C09129=1128.647,-3.756,-49.814,179.578,6.251,149.256
C09130=1128.642,-3.507,-49.827,179.579,6.255,149.256
C09131=1128.636,-3.257,-49.840,179.579,6.260,149.257
C09132=1128.632,-3.007,-49.853,179.580,6.265,149.258
C09133=1128.627,-2.758,-49.866,179.581,6.269,149.259
C09134=1128.621,-2.508,-49.879,179.581,6.274,149.260
C09135=1128.616,-2.259,-49.891,179.582,6.278,149.260
C09136=1128.611,-2.009,-49.905,179.582,6.283,149.261
C09137=1128.605,-1.760,-49.918,179.583,6.287,149.262
C09138=1128.600,-1.510,-49.930,179.583,6.291,149.263
C09139=1128.595,-1.260,-49.944,179.584,6.296,149.264
C09140=1128.590,-1.011,-49.956,179.585,6.300,149.264
C09141=1128.585,-0.761,-49.969,179.585,6.305,149.265
C09142=1128.580,-0.511,-49.982,179.586,6.310,149.266
C09143=1128.575,-0.262,-49.996,179.586,6.314,149.267
C09144=1128.569,-0.012,-50.009,179.587,6.318,149.268
C09145=1128.564,0.237,-50.022,179.587,6.323,149.269
C09146=1128.559,0.487,-50.035,179.588,6.328,149.269
C09147=1128.554,0.737,-50.048,179.588,6.332,149.270
C09148=1128.549,0.986,-50.061,179.589,6.337,149.271
C09149=1128.543,1.235,-50.075,179.589,6.341,149.272
C09150=1128.539,1.485,-50.088,179.590,6.345,149.273
C09151=1128.534,1.735,-50.100,179.590,6.350,149.274
C09152=1128.528,1.985,-50.114,179.591,6.355,149.274
C09153=1128.523,2.234,-50.126,179.591,6.360,149.275
C09154=1128.518,2.483,-50.140,179.592,6.363,149.276
C09155=1128.513,2.733,-50.153,179.592,6.368,149.277
C09156=1128.507,2.983,-50.166,179.593,6.373,149.278
C09157=1128.503,3.233,-50.179,179.593,6.377,149.279
C09158=1128.497,3.482,-50.193,179.593,6.381,149.280
C09159=1128.492,3.731,-50.206,179.594,6.386,149.280
C09160=1128.487,3.982,-50.219,179.595,6.390,149.281
C09161=1128.482,4.230,-50.233,179.595,6.395,149.282
C09162=1128.477,4.481,-50.246,179.596,6.400,149.283
C09163=1128.472,4.730,-50.259,179.596,6.404,149.284
C09164=1128.466,4.980,-50.273,179.596,6.408,149.285
C09165=1128.462,5.229,-50.286,179.597,6.413,149.285
C09166=1128.456,5.479,-50.299,179.597,6.418,149.286
C09167=1128.452,5.728,-50.313,179.597,6.422,149.287
C09168=1128.446,5.978,-50.326,179.598,6.426,149.288
C09169=1128.441,6.228,-50.339,179.599,6.431,149.289
C09170=1128.436,6.477,-50.353,179.599,6.435,149.290
C09171=1128.431,6.693,-50.364,179.599,6.439,149.291
C09172=1128.427,6.908,-50.375,179.600,6.443,149.291
C09173=1128.423,7.123,-50.387,179.600,6.447,149.292
C09174=1128.418,7.339,-50.399,179.600,6.450,149.293
C09175=1128.413,7.555,-50.410,179.601,6.455,149.293
C09176=1128.409,7.770,-50.422,179.601,6.459,149.294
C09177=1128.405,7.985,-50.434,179.601,6.462,149.295
C09178=1128.401,8.200,-50.445,179.601,6.466,149.296
C09179=1128.395,8.450,-50.459,179.602,6.470,149.296
C09180=1128.390,8.700,-50.473,179.604,6.476,149.297
C09181=1128.385,8.949,-50.485,179.605,6.480,149.298
C09182=1128.380,9.199,-50.500,179.605,6.485,149.299
C09183=1128.375,9.448,-50.512,179.606,6.490,149.300
C09184=1128.370,9.698,-50.527,179.607,6.495,149.300
C09185=1128.364,9.947,-50.540,179.608,6.500,149.301
C09186=1128.360,10.197,-50.554,179.609,6.504,149.302
C09187=1128.354,10.447,-50.567,179.609,6.509,149.303
C09188=1128.349,10.696,-50.581,179.611,6.514,149.303
C09189=1128.344,10.946,-50.594,179.612,6.518,149.304
C09190=1128.339,11.195,-50.608,179.612,6.523,149.305
C09191=1128.334,11.446,-50.621,179.613,6.528,149.306
C09192=1128.328,11.695,-50.635,179.614,6.533,149.307
C09193=1128.324,11.944,-50.649,179.615,6.537,149.307
C09194=1128.318,12.194,-50.662,179.616,6.542,149.308
C09195=1128.313,12.443,-50.676,179.617,6.546,149.309
C09196=1128.308,12.693,-50.689,179.618,6.552,149.310
C09197=1128.303,12.942,-50.703,179.619,6.556,149.310
C09198=1128.298,13.192,-50.718,179.620,6.561,149.311
C09199=1128.292,13.442,-50.731,179.621,6.565,149.312
C09200=1128.288,13.691,-50.745,179.622,6.570,149.313
C09201=1128.283,13.941,-50.759,179.623,6.575,149.313
C09202=1128.277,14.190,-50.772,179.624,6.579,149.314
C09203=1128.272,14.440,-50.786,179.625,6.584,149.315
C09204=1128.267,14.689,-50.800,179.626,6.588,149.316
C09205=1128.262,14.939,-50.814,179.627,6.593,149.316
C09206=1128.257,15.189,-50.827,179.628,6.598,149.317
C09207=1128.252,15.438,-50.841,179.629,6.603,149.318
C09208=1128.247,15.688,-50.856,179.629,6.607,149.319
C09209=1128.242,15.937,-50.870,179.630,6.612,149.319
C09210=1128.236,16.187,-50.883,179.631,6.616,149.320
C09211=1128.232,16.436,-50.897,179.632,6.621,149.321
C09212=1128.227,16.686,-50.911,179.634,6.626,149.321
C09213=1128.221,16.935,-50.925,179.635,6.630,149.322
C09214=1128.216,17.185,-50.939,179.635,6.635,149.323
C09215=1128.211,17.435,-50.953,179.636,6.639,149.324
C09216=1128.205,17.684,-50.967,179.637,6.644,149.324
C09217=1128.200,17.934,-50.981,179.639,6.649,149.325
C09218=1128.195,18.184,-50.995,179.640,6.653,149.326
C09219=1128.191,18.432,-51.009,179.641,6.658,149.326
C09220=1128.186,18.682,-51.023,179.641,6.662,149.327
C09221=1128.181,18.932,-51.037,179.642,6.667,149.328
C09222=1128.176,19.181,-51.051,179.643,6.671,149.329
C09223=1128.170,19.431,-51.065,179.645,6.676,149.329
C09224=1128.165,19.681,-51.079,179.645,6.681,149.330
C09225=1128.160,19.930,-51.093,179.647,6.685,149.331
C09226=1128.155,20.180,-51.107,179.648,6.690,149.331
C09227=1128.151,20.395,-51.120,179.649,6.694,149.332
C09228=1128.146,20.610,-51.132,179.649,6.697,149.333
C09229=1128.142,20.826,-51.144,179.651,6.701,149.333
C09230=1128.137,21.041,-51.156,179.651,6.705,149.334
C09231=1128.133,21.256,-51.168,179.652,6.709,149.335
C09232=1128.128,21.471,-51.181,179.652,6.713,149.335
C09233=1128.124,21.687,-51.192,179.654,6.717,149.336
C09234=1128.120,21.902,-51.205,179.655,6.721,149.336
C09235=1128.115,22.151,-51.220,179.656,6.725,149.337
C09236=1128.110,22.401,-51.234,179.657,6.730,149.338
C09237=1128.105,22.651,-51.248,179.658,6.734,149.338
C09238=1128.099,22.900,-51.262,179.659,6.739,149.339
C09239=1128.094,23.149,-51.276,179.660,6.743,149.340
C09240=1128.089,23.399,-51.291,179.661,6.747,149.340
C09241=1128.084,23.649,-51.305,179.662,6.752,149.341
C09242=1128.079,23.899,-51.319,179.664,6.757,149.342
C09243=1128.074,24.148,-51.334,179.664,6.761,149.343
C09244=1128.069,24.397,-51.348,179.665,6.766,149.343
C09245=1128.063,24.647,-51.363,179.666,6.770,149.344
C09246=1128.058,24.896,-51.377,179.667,6.774,149.344
C09247=1128.054,25.146,-51.392,179.668,6.779,149.345
C09248=1128.049,25.396,-51.406,179.669,6.783,149.346
C09249=1128.044,25.646,-51.420,179.670,6.787,149.346
C09250=1128.038,25.894,-51.435,179.672,6.792,149.347
C09251=1128.033,26.144,-51.449,179.673,6.797,149.348
C09252=1128.028,26.393,-51.463,179.674,6.801,149.348
C09253=1128.023,26.643,-51.478,179.675,6.805,149.349
C09254=1128.018,26.893,-51.492,179.676,6.810,149.350
C09255=1128.013,27.142,-51.507,179.677,6.814,149.351
C09256=1128.008,27.392,-51.522,179.678,6.819,149.351
C09257=1128.003,27.642,-51.536,179.679,6.823,149.352
C09258=1127.998,27.890,-51.551,179.680,6.827,149.352
C09259=1127.992,28.140,-51.566,179.681,6.832,149.353
C09260=1127.987,28.390,-51.580,179.682,6.836,149.354
C09261=1127.982,28.639,-51.594,179.684,6.841,149.354
C09262=1127.978,28.889,-51.609,179.685,6.845,149.355
C09263=1127.972,29.139,-51.624,179.686,6.850,149.356
C09264=1127.967,29.388,-51.638,179.687,6.854,149.356
C09265=1127.962,29.637,-51.653,179.688,6.858,149.357
C09266=1127.958,29.887,-51.668,179.690,6.862,149.357
C09267=1127.953,30.136,-51.683,179.691,6.867,149.358
C09268=1127.947,30.386,-51.697,179.692,6.871,149.359
C09269=1127.942,30.636,-51.712,179.693,6.875,149.359
C09270=1127.938,30.885,-51.727,179.694,6.880,149.360
C09271=1127.932,31.135,-51.742,179.695,6.884,149.361
C09272=1127.927,31.384,-51.757,179.696,6.888,149.361
C09273=1127.922,31.634,-51.771,179.698,6.893,149.362
C09274=1127.917,31.884,-51.785,179.699,6.898,149.363
C09275=1127.912,32.133,-51.801,179.700,6.902,149.363
C09276=1127.907,32.383,-51.815,179.701,6.906,149.364
C09277=1127.902,32.632,-51.830,179.702,6.910,149.365
C09278=1127.897,32.882,-51.845,179.703,6.915,149.365
C09279=1127.892,33.131,-51.860,179.704,6.919,149.366
C09280=1127.887,33.381,-51.874,179.705,6.923,149.366
C09281=1127.882,33.630,-51.890,179.707,6.927,149.367
C09282=1127.877,33.880,-51.904,179.708,6.932,149.368
C09283=1127.872,34.095,-51.917,179.709,6.936,149.368
C09284=1127.867,34.310,-51.930,179.710,6.939,149.369
C09285=1127.863,34.525,-51.943,179.711,6.943,149.369
C09286=1127.860,34.740,-51.956,179.712,6.947,149.370
C09287=1127.855,34.955,-51.969,179.713,6.950,149.370
C09288=1127.850,35.170,-51.982,179.714,6.954,149.371
C09289=1127.846,35.386,-51.994,179.715,6.958,149.371
C09290=1127.841,35.601,-52.007,179.716,6.961,149.372
C09291=1127.837,35.850,-52.022,179.717,6.965,149.372
C09292=1127.831,36.100,-52.037,179.718,6.970,149.373
C09293=1127.827,36.349,-52.052,179.719,6.974,149.374
C09294=1127.821,36.599,-52.068,179.720,6.978,149.374
C09295=1127.816,36.848,-52.082,179.721,6.983,149.375
C09296=1127.811,37.098,-52.098,179.723,6.987,149.375
C09297=1127.806,37.347,-52.113,179.724,6.991,149.376
C09298=1127.801,37.596,-52.128,179.725,6.995,149.377
C09299=1127.796,37.846,-52.142,179.726,6.999,149.377
C09300=1127.791,38.096,-52.158,179.727,7.004,149.378
C09301=1127.786,38.345,-52.173,179.729,7.008,149.378
C09302=1127.781,38.595,-52.188,179.730,7.013,149.379
C09303=1127.776,38.844,-52.203,179.731,7.017,149.380
C09304=1127.771,39.094,-52.219,179.733,7.021,149.380
C09305=1127.766,39.343,-52.234,179.734,7.025,149.381
C09306=1127.760,39.593,-52.249,179.735,7.030,149.381
C09307=1127.756,39.842,-52.264,179.736,7.034,149.382
C09308=1127.751,40.092,-52.280,179.738,7.038,149.382
C09309=1127.746,40.341,-52.295,179.739,7.042,149.383
C09310=1127.741,40.590,-52.310,179.740,7.047,149.384
C09311=1127.735,40.840,-52.326,179.741,7.051,149.384
C09312=1127.730,41.090,-52.340,179.743,7.055,149.385
C09313=1127.725,41.339,-52.356,179.744,7.059,149.385
C09314=1127.720,41.588,-52.371,179.745,7.063,149.386
C09315=1127.716,41.838,-52.387,179.746,7.067,149.386
C09316=1127.710,42.088,-52.402,179.747,7.072,149.387
C09317=1127.706,42.337,-52.417,179.748,7.076,149.388
C09318=1127.700,42.586,-52.433,179.750,7.080,149.388
C09319=1127.696,42.835,-52.448,179.751,7.084,149.389
C09320=1127.691,43.085,-52.464,179.752,7.088,149.389
C09321=1127.685,43.335,-52.479,179.754,7.092,149.390
C09322=1127.680,43.584,-52.494,179.755,7.097,149.391
C09323=1127.675,43.834,-52.509,179.756,7.101,149.391
C09324=1127.670,44.083,-52.525,179.757,7.105,149.392
C09325=1127.666,44.333,-52.540,179.758,7.109,149.392
C09326=1127.660,44.582,-52.556,179.759,7.113,149.393
C09327=1127.655,44.832,-52.571,179.761,7.117,149.393
C09328=1127.650,45.081,-52.586,179.762,7.122,149.394
C09329=1127.645,45.331,-52.602,179.764,7.126,149.394
C09330=1127.640,45.580,-52.618,179.765,7.130,149.395
C09331=1127.635,45.829,-52.634,179.766,7.134,149.396
C09332=1127.630,46.078,-52.649,179.767,7.138,149.396
C09333=1127.626,46.328,-52.665,179.768,7.142,149.397
C09334=1127.620,46.578,-52.681,179.770,7.146,149.397
C09335=1127.615,46.827,-52.696,179.771,7.151,149.398
C09336=1127.611,47.077,-52.712,179.772,7.155,149.398
C09337=1127.605,47.326,-52.727,179.774,7.159,149.399
C09338=1127.600,47.576,-52.743,179.775,7.163,149.400
C09339=1127.596,47.791,-52.757,179.776,7.166,149.400
C09340=1127.592,48.006,-52.770,179.777,7.170,149.400
C09341=1127.588,48.221,-52.783,179.778,7.173,149.401
C09342=1127.583,48.436,-52.797,179.779,7.178,149.401
C09343=1127.579,48.652,-52.811,179.780,7.181,149.402
C09344=1127.574,48.866,-52.825,179.782,7.185,149.402
C09345=1127.570,49.082,-52.838,179.783,7.188,149.403
C09346=1127.566,49.297,-52.851,179.784,7.191,149.403
C09347=1127.561,49.545,-52.867,179.785,7.195,149.404
C09348=1127.556,49.796,-52.883,179.786,7.199,149.404
C09349=1127.550,50.045,-52.899,179.787,7.204,149.405
C09350=1127.546,50.294,-52.914,179.789,7.207,149.405
C09351=1127.541,50.544,-52.930,179.790,7.212,149.406
C09352=1127.536,50.793,-52.946,179.792,7.216,149.406
C09353=1127.531,51.043,-52.962,179.793,7.220,149.407
C09354=1127.526,51.292,-52.978,179.794,7.224,149.407
C09355=1127.521,51.541,-52.994,179.795,7.228,149.408
C09356=1127.516,51.791,-53.010,179.797,7.232,149.409
C09357=1127.510,52.041,-53.025,179.798,7.236,149.409
C09358=1127.505,52.290,-53.042,179.799,7.240,149.410
C09359=1127.501,52.539,-53.057,179.801,7.245,149.410
C09360=1127.496,52.789,-53.073,179.802,7.249,149.411
C09361=1127.491,53.038,-53.089,179.803,7.253,149.411
C09362=1127.486,53.288,-53.105,179.805,7.257,149.412
C09363=1127.481,53.537,-53.121,179.806,7.261,149.412
C09364=1127.476,53.787,-53.137,179.807,7.265,149.413
C09365=1127.471,54.036,-53.153,179.809,7.269,149.413
C09366=1127.466,54.285,-53.169,179.810,7.273,149.414
C09367=1127.461,54.535,-53.185,179.811,7.277,149.415
C09368=1127.456,54.784,-53.202,179.813,7.281,149.415
C09369=1127.451,55.034,-53.217,179.814,7.286,149.416
C09370=1127.446,55.283,-53.233,179.815,7.290,149.416
C09371=1127.441,55.533,-53.250,179.817,7.293,149.416
C09372=1127.436,55.782,-53.265,179.818,7.298,149.417
C09373=1127.431,56.031,-53.282,179.820,7.302,149.418
C09374=1127.426,56.281,-53.297,179.821,7.306,149.418
C09375=1127.422,56.530,-53.314,179.822,7.310,149.419
C09376=1127.416,56.780,-53.330,179.823,7.314,149.419
C09377=1127.411,57.030,-53.347,179.825,7.318,149.420
C09378=1127.406,57.278,-53.363,179.826,7.322,149.420
C09379=1127.401,57.528,-53.379,179.828,7.326,149.421
C09380=1127.396,57.777,-53.396,179.829,7.330,149.421
C09381=1127.391,58.027,-53.411,179.830,7.335,149.422
C09382=1127.386,58.276,-53.428,179.832,7.338,149.422
C09383=1127.381,58.526,-53.444,179.833,7.342,149.423
C09384=1127.376,58.775,-53.460,179.834,7.347,149.423
C09385=1127.372,59.024,-53.477,179.836,7.351,149.424
C09386=1127.366,59.274,-53.492,179.837,7.355,149.424
C09387=1127.361,59.524,-53.510,179.839,7.359,149.425
C09388=1127.356,59.772,-53.526,179.840,7.363,149.425
C09389=1127.351,60.023,-53.542,179.841,7.367,149.426
C09390=1127.346,60.271,-53.558,179.843,7.371,149.426
C09391=1127.342,60.521,-53.575,179.844,7.374,149.427
C09392=1127.336,60.770,-53.590,179.845,7.378,149.427
C09393=1127.331,61.020,-53.608,179.847,7.382,149.428
C09394=1127.327,61.269,-53.624,179.848,7.386,149.428
C09395=1127.322,61.484,-53.638,179.849,7.390,149.429
C09396=1127.318,61.699,-53.653,179.850,7.394,149.429
C09397=1127.314,61.914,-53.667,179.852,7.397,149.430
C09398=1127.309,62.129,-53.680,179.853,7.401,149.430
C09399=1127.305,62.345,-53.694,179.854,7.404,149.431
C09400=1127.301,62.560,-53.709,179.855,7.408,149.431
C09401=1127.296,62.774,-53.723,179.856,7.411,149.431
C09402=1127.292,62.990,-53.737,179.858,7.415,149.432
C09403=1127.288,63.239,-53.754,179.859,7.419,149.432
C09404=1127.282,63.488,-53.770,179.861,7.422,149.433
C09405=1127.278,63.737,-53.787,179.862,7.427,149.433
C09406=1127.273,63.987,-53.804,179.863,7.431,149.434
C09407=1127.267,64.237,-53.820,179.865,7.435,149.434
C09408=1127.263,64.486,-53.837,179.866,7.439,149.435
C09409=1127.257,64.735,-53.854,179.868,7.443,149.435
C09410=1127.253,64.985,-53.870,179.869,7.446,149.436
C09411=1127.248,65.234,-53.887,179.870,7.450,149.436
C09412=1127.243,65.483,-53.903,179.871,7.454,149.437
C09413=1127.238,65.733,-53.920,179.873,7.458,149.437
C09414=1127.233,65.982,-53.937,179.874,7.462,149.438
C09415=1127.228,66.231,-53.953,179.876,7.466,149.438
C09416=1127.223,66.481,-53.971,179.877,7.470,149.439
C09417=1127.219,66.730,-53.987,179.878,7.474,149.439
C09418=1127.213,66.979,-54.004,179.880,7.478,149.440
C09419=1127.208,67.229,-54.021,179.881,7.482,149.440
C09420=1127.204,67.478,-54.038,179.883,7.486,149.441
C09421=1127.199,67.728,-54.054,179.884,7.490,149.441
C09422=1127.193,67.977,-54.071,179.886,7.494,149.442
C09423=1127.189,68.226,-54.088,179.887,7.498,149.442
C09424=1127.184,68.476,-54.105,179.888,7.502,149.443
C09425=1127.179,68.725,-54.121,179.890,7.506,149.443
C09426=1127.173,68.975,-54.139,179.891,7.510,149.444
C09427=1127.169,69.224,-54.155,179.893,7.514,149.444
C09428=1127.165,69.474,-54.172,179.894,7.518,149.445
C09429=1127.159,69.723,-54.189,179.896,7.522,149.445
C09430=1127.154,69.972,-54.206,179.897,7.526,149.446
C09431=1127.149,70.222,-54.223,179.898,7.531,149.446
C09432=1127.145,70.471,-54.239,179.900,7.534,149.447
C09433=1127.139,70.720,-54.257,179.902,7.538,149.447
C09434=1127.135,70.969,-54.274,179.903,7.542,149.447
C09435=1127.129,71.219,-54.291,179.904,7.547,149.448
C09436=1127.125,71.469,-54.308,179.906,7.550,149.449
C09437=1127.119,71.718,-54.325,179.907,7.554,149.449
C09438=1127.115,71.967,-54.341,179.909,7.558,149.449
C09439=1127.110,72.216,-54.359,179.909,7.562,149.450
C09440=1127.105,72.466,-54.376,179.911,7.566,149.450
C09441=1127.100,72.716,-54.393,179.913,7.570,149.451
C09442=1127.095,72.965,-54.409,179.914,7.573,149.451
C09443=1127.090,73.214,-54.427,179.915,7.578,149.452
C09444=1127.085,73.463,-54.444,179.917,7.582,149.452
C09445=1127.080,73.713,-54.461,179.918,7.586,149.453
C09446=1127.075,73.963,-54.479,179.920,7.589,149.453
C09447=1127.070,74.211,-54.496,179.921,7.594,149.454
C09448=1127.065,74.461,-54.513,179.923,7.598,149.454
C09449=1127.061,74.710,-54.530,179.924,7.602,149.455
C09450=1127.056,74.959,-54.548,179.926,7.605,149.455
C09451=1127.051,75.175,-54.562,179.928,7.609,149.456
C09452=1127.047,75.390,-54.577,179.928,7.612,149.456
C09453=1127.043,75.605,-54.592,179.929,7.616,149.456
C09454=1127.038,75.819,-54.606,179.931,7.620,149.457
C09455=1127.034,76.034,-54.621,179.932,7.623,149.457
C09456=1127.030,76.249,-54.636,179.934,7.627,149.458
C09457=1127.026,76.464,-54.651,179.934,7.630,149.458
C09458=1127.021,76.679,-54.666,179.936,7.634,149.459
C09459=1127.017,76.928,-54.684,179.937,7.637,149.459
C09460=1127.012,77.178,-54.701,179.938,7.640,149.460
C09461=1127.007,77.427,-54.719,179.939,7.644,149.460
C09462=1127.002,77.677,-54.735,179.940,7.648,149.461
C09463=1126.997,77.925,-54.753,179.941,7.652,149.461
C09464=1126.992,78.175,-54.770,179.942,7.655,149.462
C09465=1126.987,78.424,-54.787,179.943,7.659,149.462
C09466=1126.982,78.674,-54.805,179.944,7.662,149.463
C09467=1126.977,78.923,-54.822,179.945,7.667,149.464
C09468=1126.972,79.173,-54.840,179.946,7.670,149.464
C09469=1126.968,79.422,-54.857,179.947,7.674,149.465
C09470=1126.963,79.671,-54.875,179.948,7.678,149.465
C09471=1126.958,79.921,-54.892,179.949,7.681,149.466
C09472=1126.953,80.170,-54.909,179.950,7.685,149.466
C09473=1126.948,80.419,-54.927,179.951,7.689,149.467
C09474=1126.943,80.669,-54.945,179.952,7.692,149.467
C09475=1126.938,80.918,-54.963,179.953,7.696,149.468
C09476=1126.933,81.168,-54.980,179.954,7.701,149.468
C09477=1126.928,81.416,-54.997,179.955,7.704,149.469
C09478=1126.923,81.666,-55.014,179.957,7.708,149.469
C09479=1126.918,81.915,-55.032,179.957,7.711,149.470
C09480=1126.913,82.164,-55.050,179.959,7.715,149.470
C09481=1126.909,82.414,-55.067,179.960,7.719,149.471
C09482=1126.904,82.663,-55.085,179.961,7.722,149.471
C09483=1126.899,82.912,-55.103,179.962,7.727,149.472
C09484=1126.894,83.162,-55.120,179.964,7.731,149.472
C09485=1126.889,83.411,-55.138,179.965,7.734,149.473
C09486=1126.884,83.660,-55.156,179.966,7.738,149.474
C09487=1126.879,83.910,-55.173,179.968,7.742,149.474
C09488=1126.875,84.159,-55.191,179.969,7.746,149.475
C09489=1126.870,84.408,-55.209,179.970,7.749,149.475
C09490=1126.864,84.658,-55.226,179.971,7.753,149.475
C09491=1126.860,84.907,-55.244,179.972,7.757,149.476
C09492=1126.855,85.156,-55.262,179.973,7.761,149.477
C09493=1126.849,85.406,-55.279,179.975,7.764,149.477
C09494=1126.844,85.655,-55.297,179.976,7.769,149.478
C09495=1126.840,85.904,-55.315,179.978,7.773,149.478
C09496=1126.836,86.154,-55.333,179.979,7.776,149.478
C09497=1126.831,86.403,-55.351,179.980,7.780,149.479
C09498=1126.826,86.653,-55.368,179.981,7.784,149.480
C09499=1126.821,86.902,-55.386,179.983,7.788,149.480
C09500=1126.816,87.151,-55.404,179.985,7.792,149.480
C09501=1126.811,87.400,-55.422,179.986,7.796,149.481
C09502=1126.806,87.649,-55.440,179.987,7.800,149.481
C09503=1126.801,87.899,-55.457,179.988,7.803,149.482
C09504=1126.796,88.148,-55.475,179.990,7.807,149.482
C09505=1126.791,88.398,-55.493,179.991,7.811,149.483
C09506=1126.786,88.647,-55.511,179.993,7.815,149.483
C09507=1126.782,88.862,-55.527,179.994,7.818,149.484
C09508=1126.778,89.076,-55.542,179.995,7.822,149.484
C09509=1126.774,89.291,-55.557,179.997,7.825,149.484
C09510=1126.770,89.506,-55.573,179.998,7.828,149.485
C09511=1126.765,89.721,-55.589,179.999,7.832,149.485
C09512=1126.761,89.936,-55.605,-180.000,7.835,149.486
C09513=1126.757,90.151,-55.620,-179.998,7.839,149.486
C09514=1126.753,90.366,-55.635,-179.997,7.842,149.487
C09515=1126.748,90.615,-55.653,-179.996,7.846,149.487
C09516=1126.743,90.864,-55.671,-179.994,7.850,149.487
C09517=1126.738,91.113,-55.689,-179.993,7.854,149.488
C09518=1126.733,91.362,-55.707,-179.991,7.857,149.488
C09519=1126.729,91.611,-55.725,-179.989,7.861,149.489
C09520=1126.724,91.861,-55.744,-179.988,7.865,149.489
C09521=1126.719,92.111,-55.762,-179.986,7.869,149.490
C09522=1126.714,92.360,-55.780,-179.985,7.873,149.490
C09523=1126.709,92.609,-55.798,-179.983,7.877,149.490
C09524=1126.704,92.858,-55.816,-179.981,7.881,149.491
C09525=1126.699,93.108,-55.834,-179.980,7.885,149.491
C09526=1126.695,93.357,-55.852,-179.978,7.889,149.492
C09527=1126.690,93.607,-55.870,-179.977,7.892,149.492
C09528=1126.685,93.855,-55.889,-179.975,7.896,149.493
C09529=1126.679,94.105,-55.908,-179.973,7.900,149.493
C09530=1126.675,94.354,-55.926,-179.972,7.904,149.493
C09531=1126.670,94.604,-55.944,-179.970,7.909,149.494
C09532=1126.665,94.853,-55.962,-179.968,7.913,149.494
C09533=1126.660,95.102,-55.980,-179.966,7.917,149.495
C09534=1126.656,95.351,-55.999,-179.965,7.920,149.495
C09535=1126.651,95.601,-56.018,-179.963,7.924,149.496
C09536=1126.646,95.850,-56.036,-179.961,7.928,149.496
C09537=1126.641,96.099,-56.054,-179.959,7.932,149.496
C09538=1126.636,96.348,-56.072,-179.957,7.936,149.497
C09539=1126.632,96.598,-56.091,-179.956,7.940,149.497
C09540=1126.626,96.847,-56.109,-179.954,7.944,149.498
C09541=1126.621,97.096,-56.127,-179.952,7.948,149.498
C09542=1126.617,97.345,-56.145,-179.950,7.952,149.498
C09543=1126.612,97.595,-56.165,-179.949,7.955,149.499
C09544=1126.607,97.844,-56.183,-179.947,7.960,149.499
C09545=1126.602,98.093,-56.201,-179.945,7.964,149.499
C09546=1126.597,98.342,-56.219,-179.943,7.968,149.500
C09547=1126.592,98.592,-56.238,-179.941,7.971,149.500
C09548=1126.587,98.841,-56.256,-179.939,7.976,149.501
C09549=1126.583,99.090,-56.275,-179.937,7.980,149.501
C09550=1126.578,99.340,-56.294,-179.935,7.983,149.501
C09551=1126.573,99.589,-56.313,-179.933,7.987,149.501
C09552=1126.568,99.838,-56.331,-179.931,7.992,149.502
C09553=1126.563,100.088,-56.350,-179.930,7.996,149.502
C09554=1126.559,100.336,-56.368,-179.927,7.999,149.502
C09555=1126.554,100.586,-56.386,-179.926,8.003,149.503
C09556=1126.549,100.835,-56.406,-179.923,8.007,149.503
C09557=1126.544,101.084,-56.424,-179.922,8.011,149.504
C09558=1126.539,101.333,-56.443,-179.920,8.015,149.504
C09559=1126.534,101.583,-56.462,-179.917,8.019,149.504
C09560=1126.530,101.832,-56.480,-179.916,8.023,149.505
C09561=1126.525,102.082,-56.499,-179.914,8.027,149.505
C09562=1126.520,102.330,-56.518,-179.911,8.031,149.505
C09563=1126.515,102.545,-56.534,-179.910,8.034,149.505
C09564=1126.511,102.760,-56.550,-179.908,8.038,149.506
C09565=1126.507,102.975,-56.566,-179.906,8.041,149.506
C09566=1126.503,103.189,-56.582,-179.904,8.045,149.506
C09567=1126.499,103.404,-56.599,-179.902,8.048,149.507
C09568=1126.495,103.619,-56.615,-179.901,8.051,149.507
C09569=1126.491,103.834,-56.632,-179.899,8.055,149.507
C09570=1126.487,104.048,-56.647,-179.897,8.058,149.507
C09571=1126.482,104.298,-56.667,-179.895,8.062,149.507
C09572=1126.477,104.547,-56.685,-179.892,8.066,149.508
C09573=1126.472,104.797,-56.704,-179.890,8.070,149.508
C09574=1126.468,105.045,-56.723,-179.888,8.074,149.508
C09575=1126.462,105.294,-56.742,-179.886,8.078,149.509
C09576=1126.458,105.544,-56.761,-179.884,8.082,149.509
C09577=1126.453,105.793,-56.780,-179.881,8.086,149.509
C09578=1126.448,106.042,-56.799,-179.879,8.089,149.509
C09579=1126.443,106.291,-56.818,-179.877,8.094,149.510
C09580=1126.438,106.541,-56.837,-179.875,8.097,149.510
C09581=1126.434,106.790,-56.856,-179.872,8.102,149.510
C09582=1126.429,107.039,-56.875,-179.870,8.105,149.510
C09583=1126.424,107.288,-56.894,-179.867,8.110,149.511
C09584=1126.419,107.538,-56.913,-179.865,8.113,149.511
C09585=1126.414,107.787,-56.932,-179.863,8.117,149.511
C09586=1126.410,108.036,-56.951,-179.861,8.121,149.511
C09587=1126.404,108.285,-56.971,-179.858,8.125,149.512
C09588=1126.400,108.535,-56.990,-179.856,8.129,149.512
C09589=1126.395,108.783,-57.009,-179.853,8.133,149.512
C09590=1126.390,109.033,-57.029,-179.851,8.136,149.512
C09591=1126.386,109.282,-57.048,-179.849,8.141,149.512
C09592=1126.381,109.532,-57.066,-179.846,8.144,149.513
C09593=1126.376,109.781,-57.086,-179.844,8.148,149.513
C09594=1126.371,110.030,-57.105,-179.841,8.153,149.513
C09595=1126.367,110.279,-57.124,-179.839,8.156,149.513
C09596=1126.361,110.528,-57.144,-179.836,8.160,149.514
C09597=1126.357,110.778,-57.163,-179.834,8.164,149.514
C09598=1126.352,111.027,-57.183,-179.832,8.168,149.514
C09599=1126.347,111.276,-57.202,-179.830,8.172,149.514
C09600=1126.342,111.525,-57.221,-179.828,8.174,149.514
C09601=1126.337,111.774,-57.241,-179.826,8.178,149.515
C09602=1126.332,112.024,-57.260,-179.824,8.182,149.515
C09603=1126.328,112.273,-57.280,-179.822,8.185,149.515
C09604=1126.323,112.521,-57.299,-179.820,8.189,149.516
C09605=1126.319,112.771,-57.319,-179.818,8.192,149.516
C09606=1126.313,113.020,-57.338,-179.817,8.196,149.516
C09607=1126.308,113.269,-57.358,-179.815,8.200,149.516
C09608=1126.304,113.519,-57.378,-179.812,8.203,149.517
C09609=1126.298,113.768,-57.397,-179.810,8.207,149.517
C09610=1126.294,114.017,-57.416,-179.809,8.211,149.517
C09611=1126.290,114.267,-57.436,-179.807,8.214,149.518
C09612=1126.285,114.515,-57.456,-179.805,8.218,149.518
C09613=1126.280,114.764,-57.475,-179.803,8.221,149.518
C09614=1126.275,115.014,-57.495,-179.801,8.224,149.518
C09615=1126.270,115.263,-57.514,-179.800,8.228,149.519
C09616=1126.265,115.512,-57.534,-179.798,8.231,149.519
C09617=1126.261,115.761,-57.554,-179.795,8.235,149.519
C09618=1126.256,116.010,-57.573,-179.793,8.238,149.519
C09619=1126.252,116.225,-57.590,-179.792,8.241,149.519
C09620=1126.247,116.439,-57.607,-179.790,8.244,149.520
C09621=1126.244,116.655,-57.624,-179.788,8.247,149.520
C09622=1126.240,116.869,-57.642,-179.787,8.250,149.520
C09623=1126.235,117.083,-57.658,-179.786,8.253,149.520
C09624=1126.231,117.299,-57.675,-179.784,8.256,149.521
C09625=1126.227,117.513,-57.692,-179.782,8.259,149.521
C09626=1126.223,117.727,-57.710,-179.781,8.262,149.521
C09627=1126.218,117.976,-57.729,-179.779,8.265,149.521
C09628=1126.213,118.226,-57.749,-179.777,8.269,149.522
C09629=1126.209,118.475,-57.769,-179.775,8.272,149.522
C09630=1126.204,118.724,-57.789,-179.773,8.276,149.522
C09631=1126.199,118.973,-57.808,-179.771,8.279,149.522
C09632=1126.194,119.222,-57.828,-179.770,8.283,149.523
C09633=1126.189,119.472,-57.848,-179.768,8.286,149.523
C09634=1126.185,119.721,-57.868,-179.766,8.289,149.523
C09635=1126.180,119.970,-57.888,-179.764,8.293,149.523
C09636=1126.175,120.219,-57.907,-179.762,8.296,149.524
C09637=1126.170,120.468,-57.928,-179.760,8.300,149.524
C09638=1126.166,120.718,-57.947,-179.758,8.303,149.524
C09639=1126.161,120.967,-57.968,-179.756,8.307,149.525
C09640=1126.156,121.216,-57.987,-179.754,8.310,149.525
C09641=1126.151,121.464,-58.007,-179.753,8.313,149.525
C09642=1126.147,121.714,-58.027,-179.751,8.317,149.525
C09643=1126.142,121.963,-58.047,-179.749,8.320,149.526
C09644=1126.137,122.213,-58.067,-179.747,8.324,149.526
C09645=1126.133,122.462,-58.088,-179.746,8.326,149.526
C09646=1126.127,122.711,-58.107,-179.744,8.330,149.527
C09647=1126.123,122.960,-58.128,-179.742,8.334,149.527
C09648=1126.118,123.209,-58.147,-179.740,8.337,149.527
C09649=1126.113,123.458,-58.168,-179.738,8.340,149.527
C09650=1126.109,123.707,-58.188,-179.736,8.343,149.527
C09651=1126.104,123.957,-58.208,-179.735,8.347,149.528
C09652=1126.099,124.205,-58.228,-179.733,8.351,149.528
C09653=1126.094,124.455,-58.248,-179.731,8.354,149.528
C09654=1126.089,124.704,-58.268,-179.729,8.357,149.529
C09655=1126.085,124.953,-58.289,-179.727,8.361,149.529
C09656=1126.080,125.202,-58.308,-179.726,8.364,149.529
C09657=1126.076,125.451,-58.329,-179.724,8.367,149.529
C09658=1126.071,125.700,-58.349,-179.722,8.371,149.530
C09659=1126.066,125.950,-58.369,-179.721,8.373,149.530
C09660=1126.061,126.199,-58.390,-179.719,8.377,149.530
C09661=1126.057,126.448,-58.410,-179.717,8.381,149.531
C09662=1126.052,126.696,-58.430,-179.715,8.383,149.531
C09663=1126.046,126.946,-58.450,-179.713,8.387,149.531
C09664=1126.042,127.195,-58.471,-179.712,8.391,149.531
C09665=1126.037,127.444,-58.491,-179.710,8.394,149.532
C09666=1126.033,127.693,-58.512,-179.708,8.397,149.532
C09667=1126.027,127.943,-58.532,-179.706,8.401,149.532
C09668=1126.023,128.192,-58.552,-179.705,8.404,149.533
C09669=1126.019,128.441,-58.573,-179.703,8.407,149.533
C09670=1126.014,128.690,-58.593,-179.701,8.411,149.533
C09671=1126.009,128.939,-58.614,-179.700,8.413,149.533
C09672=1126.004,129.188,-58.634,-179.698,8.417,149.534
C09673=1126.000,129.437,-58.654,-179.696,8.421,149.534
C09674=1125.995,129.687,-58.675,-179.694,8.423,149.534
C09675=1125.990,129.900,-58.692,-179.693,8.426,149.534
C09676=1125.987,130.115,-58.710,-179.691,8.430,149.535
C09677=1125.983,130.330,-58.727,-179.690,8.433,149.535
C09678=1125.978,130.545,-58.746,-179.688,8.435,149.535
C09679=1125.974,130.759,-58.763,-179.687,8.438,149.535
C09680=1125.970,130.973,-58.781,-179.686,8.441,149.536
C09681=1125.966,131.189,-58.798,-179.684,8.444,149.536
C09682=1125.962,131.402,-58.816,-179.683,8.446,149.536
C09683=1125.957,131.651,-58.836,-179.681,8.450,149.536
C09684=1125.952,131.901,-58.857,-179.679,8.454,149.537
C09685=1125.947,132.150,-58.878,-179.678,8.456,149.537
C09686=1125.943,132.399,-58.898,-179.675,8.460,149.537
C09687=1125.938,132.648,-58.919,-179.674,8.463,149.538
C09688=1125.934,132.897,-58.940,-179.672,8.466,149.538
C09689=1125.929,133.147,-58.961,-179.670,8.470,149.538
C09690=1125.924,133.396,-58.981,-179.669,8.473,149.538
C09691=1125.920,133.645,-59.001,-179.667,8.477,149.539
C09692=1125.915,133.894,-59.022,-179.666,8.479,149.539
C09693=1125.910,134.143,-59.043,-179.664,8.483,149.539
C09694=1125.905,134.392,-59.064,-179.663,8.486,149.540
C09695=1125.901,134.641,-59.084,-179.661,8.490,149.540
C09696=1125.896,134.890,-59.105,-179.659,8.493,149.540
C09697=1125.891,135.139,-59.125,-179.658,8.496,149.540
C09698=1125.886,135.388,-59.147,-179.656,8.500,149.541
C09699=1125.882,135.637,-59.167,-179.654,8.502,149.541
C09700=1125.877,135.886,-59.188,-179.652,8.506,149.541
C09701=1125.872,136.135,-59.209,-179.651,8.509,149.542
C09702=1125.867,136.384,-59.230,-179.649,8.513,149.542
C09703=1125.863,136.633,-59.250,-179.648,8.516,149.542
C09704=1125.858,136.883,-59.271,-179.646,8.519,149.543
C09705=1125.854,137.132,-59.292,-179.644,8.523,149.543
C09706=1125.849,137.381,-59.313,-179.643,8.526,149.543
C09707=1125.844,137.630,-59.334,-179.641,8.529,149.544
C09708=1125.839,137.879,-59.355,-179.640,8.532,149.544
C09709=1125.834,138.128,-59.376,-179.638,8.536,149.544
C09710=1125.830,138.377,-59.397,-179.637,8.539,149.545
C09711=1125.825,138.626,-59.418,-179.635,8.542,149.545
C09712=1125.821,138.876,-59.439,-179.634,8.545,149.545
C09713=1125.816,139.125,-59.460,-179.632,8.549,149.546
C09714=1125.811,139.373,-59.481,-179.631,8.552,149.546
C09715=1125.806,139.622,-59.502,-179.629,8.556,149.546
C09716=1125.801,139.872,-59.523,-179.628,8.559,149.547
C09717=1125.797,140.121,-59.543,-179.626,8.562,149.547
C09718=1125.792,140.370,-59.565,-179.625,8.565,149.547
C09719=1125.787,140.619,-59.586,-179.623,8.569,149.548
C09720=1125.783,140.868,-59.606,-179.622,8.572,149.548
C09721=1125.778,141.117,-59.628,-179.619,8.575,149.548
C09722=1125.773,141.366,-59.649,-179.618,8.578,149.549
C09723=1125.768,141.615,-59.669,-179.616,8.582,149.549
C09724=1125.764,141.864,-59.691,-179.615,8.585,149.549
C09725=1125.759,142.114,-59.712,-179.613,8.588,149.550
C09726=1125.755,142.362,-59.733,-179.612,8.592,149.550
C09727=1125.750,142.611,-59.754,-179.611,8.595,149.550
C09728=1125.744,142.860,-59.775,-179.609,8.598,149.551
C09729=1125.741,143.109,-59.797,-179.608,8.602,149.551
C09730=1125.736,143.359,-59.818,-179.606,8.605,149.551
C09731=1125.732,143.573,-59.837,-179.605,8.608,149.552
C09732=1125.728,143.787,-59.855,-179.604,8.610,149.552
C09733=1125.724,144.002,-59.873,-179.602,8.613,149.552
C09734=1125.719,144.216,-59.890,-179.601,8.616,149.553
C09735=1125.715,144.430,-59.909,-179.600,8.619,149.553
C09736=1125.712,144.645,-59.927,-179.599,8.622,149.553
C09737=1125.707,144.859,-59.946,-179.597,8.625,149.553
C09738=1125.703,145.074,-59.965,-179.596,8.628,149.554
C09739=1125.699,145.323,-59.985,-179.593,8.632,149.554
C09740=1125.694,145.572,-60.007,-179.590,8.636,149.554
C09741=1125.689,145.821,-60.028,-179.588,8.640,149.554
C09742=1125.684,146.070,-60.050,-179.586,8.644,149.555
C09743=1125.680,146.319,-60.070,-179.583,8.648,149.555
C09744=1125.676,146.568,-60.092,-179.581,8.652,149.555
C09745=1125.671,146.817,-60.113,-179.578,8.655,149.555
C09746=1125.666,147.066,-60.135,-179.575,8.660,149.555
C09747=1125.661,147.315,-60.157,-179.573,8.663,149.556
C09748=1125.656,147.565,-60.178,-179.570,8.667,149.556
C09749=1125.651,147.813,-60.200,-179.568,8.671,149.556
C09750=1125.648,148.062,-60.221,-179.565,8.675,149.556
C09751=1125.643,148.312,-60.242,-179.562,8.679,149.556
C09752=1125.638,148.560,-60.264,-179.560,8.683,149.557
C09753=1125.633,148.810,-60.286,-179.557,8.686,149.557
C09754=1125.628,149.059,-60.307,-179.555,8.690,149.557
C09755=1125.623,149.307,-60.328,-179.552,8.694,149.557
C09756=1125.619,149.557,-60.350,-179.550,8.697,149.557
C09757=1125.614,149.805,-60.372,-179.547,8.702,149.557
C09758=1125.609,150.054,-60.394,-179.545,8.705,149.558
C09759=1125.605,150.304,-60.415,-179.542,8.709,149.558
C09760=1125.600,150.553,-60.437,-179.540,8.712,149.558
C09761=1125.595,150.801,-60.458,-179.537,8.717,149.558
C09762=1125.591,151.051,-60.481,-179.534,8.720,149.558
C09763=1125.586,151.299,-60.502,-179.532,8.724,149.558
C09764=1125.581,151.549,-60.524,-179.529,8.727,149.558
C09765=1125.577,151.798,-60.545,-179.527,8.731,149.559
C09766=1125.572,152.047,-60.567,-179.524,8.735,149.559
C09767=1125.567,152.296,-60.589,-179.522,8.738,149.559
C09768=1125.563,152.545,-60.611,-179.519,8.742,149.559
C09769=1125.558,152.794,-60.633,-179.517,8.745,149.559
C09770=1125.553,153.043,-60.654,-179.515,8.749,149.559
C09771=1125.549,153.292,-60.676,-179.511,8.753,149.559
C09772=1125.544,153.540,-60.698,-179.509,8.756,149.560
C09773=1125.540,153.790,-60.720,-179.507,8.759,149.560
C09774=1125.535,154.038,-60.742,-179.504,8.764,149.560
C09775=1125.530,154.287,-60.764,-179.502,8.767,149.560
C09776=1125.525,154.537,-60.786,-179.499,8.770,149.560
C09777=1125.520,154.785,-60.808,-179.496,8.774,149.560
C09778=1125.516,155.035,-60.830,-179.494,8.778,149.560
C09779=1125.511,155.283,-60.852,-179.492,8.781,149.560
C09780=1125.507,155.533,-60.874,-179.489,8.785,149.561
C09781=1125.502,155.781,-60.895,-179.486,8.788,149.561
C09782=1125.498,156.031,-60.917,-179.484,8.792,149.561
C09783=1125.493,156.279,-60.940,-179.482,8.795,149.561
C09784=1125.488,156.528,-60.962,-179.479,8.799,149.561
C09785=1125.483,156.777,-60.984,-179.477,8.802,149.561
C09786=1125.479,157.026,-61.006,-179.474,8.805,149.561
C09787=1125.475,157.241,-61.025,-179.472,8.809,149.561
C09788=1125.471,157.455,-61.044,-179.470,8.811,149.562
C09789=1125.467,157.669,-61.063,-179.468,8.814,149.562
C09790=1125.463,157.884,-61.083,-179.466,8.818,149.562
C09791=1125.459,158.098,-61.102,-179.464,8.820,149.562
C09792=1125.455,158.312,-61.121,-179.461,8.823,149.562
C09793=1125.451,158.526,-61.140,-179.460,8.826,149.562
C09794=1125.447,158.741,-61.159,-179.457,8.829,149.562
C09795=1125.443,158.990,-61.181,-179.455,8.832,149.562
C09796=1125.437,159.239,-61.204,-179.453,8.835,149.562
C09797=1125.433,159.488,-61.226,-179.450,8.839,149.562
C09798=1125.429,159.737,-61.248,-179.448,8.842,149.563
C09799=1125.423,159.986,-61.271,-179.445,8.846,149.563
C09800=1125.419,160.235,-61.293,-179.442,8.849,149.563
C09801=1125.415,160.483,-61.315,-179.440,8.853,149.563
C09802=1125.410,160.733,-61.338,-179.438,8.856,149.563
C09803=1125.406,160.982,-61.360,-179.435,8.859,149.563
C09804=1125.401,161.230,-61.382,-179.433,8.862,149.563
C09805=1125.396,161.480,-61.405,-179.431,8.865,149.563
C09806=1125.392,161.729,-61.428,-179.428,8.868,149.563
C09807=1125.387,161.977,-61.449,-179.426,8.872,149.564
C09808=1125.382,162.226,-61.473,-179.423,8.875,149.564
C09809=1125.378,162.476,-61.495,-179.421,8.878,149.564
C09810=1125.373,162.724,-61.517,-179.419,8.882,149.564
C09811=1125.368,162.973,-61.540,-179.416,8.885,149.564
C09812=1125.364,163.222,-61.562,-179.414,8.888,149.564
C09813=1125.359,163.471,-61.585,-179.411,8.891,149.564
C09814=1125.355,163.720,-61.607,-179.409,8.894,149.564
C09815=1125.350,163.969,-61.630,-179.407,8.898,149.564
C09816=1125.345,164.217,-61.653,-179.404,8.901,149.564
C09817=1125.341,164.467,-61.675,-179.402,8.904,149.564
C09818=1125.336,164.716,-61.698,-179.399,8.907,149.564
C09819=1125.332,164.965,-61.720,-179.397,8.910,149.565
C09820=1125.327,165.213,-61.743,-179.395,8.914,149.565
C09821=1125.323,165.462,-61.766,-179.392,8.917,149.565
C09822=1125.318,165.712,-61.788,-179.390,8.920,149.565
C09823=1125.313,165.960,-61.811,-179.387,8.923,149.565
C09824=1125.308,166.209,-61.834,-179.385,8.927,149.565
C09825=1125.303,166.459,-61.857,-179.383,8.930,149.565
C09826=1125.299,166.707,-61.880,-179.380,8.933,149.565
C09827=1125.294,166.956,-61.903,-179.378,8.936,149.565
C09828=1125.290,167.205,-61.925,-179.376,8.939,149.565
C09829=1125.285,167.454,-61.948,-179.374,8.942,149.565
C09830=1125.281,167.703,-61.971,-179.371,8.945,149.566
C09831=1125.276,167.952,-61.993,-179.369,8.948,149.566
C09832=1125.271,168.201,-62.016,-179.367,8.951,149.566
C09833=1125.267,168.449,-62.039,-179.364,8.955,149.566
C09834=1125.262,168.698,-62.062,-179.361,8.958,149.566
C09835=1125.258,168.947,-62.085,-179.359,8.961,149.566
C09836=1125.253,169.196,-62.107,-179.357,8.963,149.566
C09837=1125.248,169.445,-62.131,-179.355,8.967,149.566
C09838=1125.244,169.694,-62.154,-179.352,8.970,149.566
C09839=1125.239,169.943,-62.177,-179.350,8.973,149.566
C09840=1125.235,170.192,-62.200,-179.348,8.976,149.566
C09841=1125.230,170.441,-62.222,-179.345,8.979,149.566
C09842=1125.225,170.690,-62.245,-179.344,8.982,149.567
C09843=1125.222,170.904,-62.266,-179.341,8.985,149.567
C09844=1125.217,171.118,-62.285,-179.339,8.988,149.567
C09845=1125.213,171.332,-62.305,-179.338,8.990,149.567
C09846=1125.210,171.546,-62.325,-179.336,8.992,149.567
C09847=1125.205,171.761,-62.345,-179.334,8.996,149.567
C09848=1125.202,171.975,-62.365,-179.332,8.998,149.567
C09849=1125.197,172.189,-62.385,-179.330,9.000,149.567
C09850=1125.194,172.403,-62.405,-179.328,9.003,149.567
C09851=1125.189,172.652,-62.428,-179.326,9.006,149.567
C09852=1125.185,172.901,-62.451,-179.323,9.009,149.567
C09853=1125.180,173.150,-62.474,-179.321,9.012,149.567
C09854=1125.175,173.399,-62.497,-179.319,9.015,149.568
C09855=1125.171,173.648,-62.521,-179.317,9.018,149.568
C09856=1125.167,173.897,-62.543,-179.314,9.021,149.568
C09857=1125.162,174.146,-62.567,-179.312,9.024,149.568
C09858=1125.157,174.394,-62.590,-179.310,9.027,149.568
C09859=1125.152,174.643,-62.613,-179.308,9.030,149.568
C09860=1125.147,174.892,-62.637,-179.306,9.033,149.568
C09861=1125.143,175.141,-62.659,-179.304,9.036,149.568
C09862=1125.139,175.390,-62.683,-179.301,9.039,149.568
C09863=1125.134,175.639,-62.706,-179.299,9.042,149.568
C09864=1125.130,175.887,-62.730,-179.297,9.045,149.569
C09865=1125.125,176.136,-62.753,-179.295,9.048,149.569
C09866=1125.120,176.385,-62.777,-179.293,9.050,149.569
C09867=1125.116,176.634,-62.800,-179.290,9.054,149.569
C09868=1125.112,176.883,-62.823,-179.288,9.057,149.569
C09869=1125.107,177.132,-62.846,-179.286,9.059,149.569
C09870=1125.102,177.381,-62.870,-179.284,9.062,149.569
C09871=1125.098,177.629,-62.894,-179.282,9.066,149.569
C09872=1125.093,177.879,-62.917,-179.280,9.068,149.569
C09873=1125.088,178.128,-62.940,-179.277,9.071,149.569
C09874=1125.084,178.377,-62.964,-179.275,9.075,149.570
C09875=1125.079,178.625,-62.988,-179.273,9.077,149.570
C09876=1125.075,178.874,-63.011,-179.271,9.081,149.570
C09877=1125.071,179.123,-63.034,-179.269,9.083,149.570
C09878=1125.066,179.372,-63.057,-179.267,9.086,149.570
C09879=1125.062,179.620,-63.081,-179.264,9.090,149.570
C09880=1125.057,179.869,-63.105,-179.261,9.093,149.570
C09881=1125.052,180.118,-63.128,-179.258,9.097,149.570
C09882=1125.048,180.367,-63.152,-179.255,9.100,149.570
C09883=1125.043,180.616,-63.176,-179.252,9.104,149.570
C09884=1125.038,180.865,-63.199,-179.249,9.107,149.570
C09885=1125.034,181.113,-63.223,-179.246,9.109,149.570
C09886=1125.029,181.362,-63.246,-179.243,9.113,149.570
C09887=1125.025,181.611,-63.270,-179.241,9.116,149.570
C09888=1125.020,181.860,-63.294,-179.238,9.120,149.570
C09889=1125.015,182.109,-63.317,-179.235,9.122,149.570
C09890=1125.011,182.357,-63.341,-179.232,9.126,149.570
C09891=1125.006,182.606,-63.365,-179.230,9.129,149.570
C09892=1125.002,182.856,-63.390,-179.227,9.132,149.570
C09893=1124.997,183.105,-63.413,-179.224,9.135,149.570
C09894=1124.993,183.353,-63.437,-179.222,9.138,149.570
C09895=1124.988,183.602,-63.460,-179.219,9.141,149.570
C09896=1124.984,183.850,-63.485,-179.216,9.144,149.570
C09897=1124.979,184.099,-63.508,-179.214,9.148,149.570
C09898=1124.975,184.348,-63.532,-179.211,9.150,149.570
C09899=1124.971,184.562,-63.553,-179.208,9.153,149.570
C09900=1124.966,184.776,-63.573,-179.207,9.156,149.570
C09901=1124.963,184.990,-63.594,-179.205,9.158,149.570
C09902=1124.959,185.205,-63.615,-179.202,9.161,149.570
C09903=1124.955,185.418,-63.635,-179.200,9.163,149.570
C09904=1124.951,185.633,-63.656,-179.198,9.166,149.570
C09905=1124.947,185.847,-63.676,-179.195,9.169,149.570
C09906=1124.944,186.061,-63.697,-179.194,9.171,149.570
C09907=1124.939,186.310,-63.721,-179.191,9.174,149.570
C09908=1124.934,186.558,-63.745,-179.188,9.177,149.570
C09909=1124.930,186.807,-63.770,-179.187,9.179,149.570
C09910=1124.925,187.056,-63.793,-179.184,9.183,149.570
C09911=1124.921,187.305,-63.817,-179.182,9.186,149.570
C09912=1124.916,187.553,-63.841,-179.179,9.189,149.570
C09913=1124.911,187.803,-63.865,-179.177,9.191,149.570
C09914=1124.907,188.051,-63.889,-179.175,9.194,149.570
C09915=1124.903,188.300,-63.914,-179.172,9.197,149.570
C09916=1124.898,188.549,-63.938,-179.170,9.200,149.570
C09917=1124.893,188.797,-63.962,-179.168,9.203,149.570
C09918=1124.889,189.046,-63.986,-179.166,9.205,149.570
C09919=1124.885,189.295,-64.010,-179.163,9.208,149.571
C09920=1124.880,189.544,-64.035,-179.161,9.210,149.571
C09921=1124.875,189.793,-64.059,-179.159,9.214,149.571
C09922=1124.871,190.041,-64.083,-179.157,9.216,149.571
C09923=1124.866,190.291,-64.107,-179.154,9.219,149.571
C09924=1124.862,190.539,-64.131,-179.152,9.221,149.571
C09925=1124.857,190.788,-64.155,-179.150,9.224,149.571
C09926=1124.852,191.037,-64.180,-179.148,9.227,149.571
C09927=1124.848,191.286,-64.205,-179.147,9.230,149.571
C09928=1124.844,191.534,-64.229,-179.144,9.233,149.571
C09929=1124.839,191.783,-64.253,-179.142,9.235,149.571
C09930=1124.834,192.031,-64.277,-179.140,9.237,149.571
C09931=1124.830,192.281,-64.302,-179.138,9.241,149.571
C09932=1124.825,192.529,-64.327,-179.136,9.243,149.571
C09933=1124.821,192.777,-64.351,-179.134,9.245,149.571
C09934=1124.816,193.026,-64.375,-179.133,9.248,149.572
C09935=1124.812,193.276,-64.399,-179.130,9.251,149.572
C09936=1124.807,193.525,-64.424,-179.128,9.254,149.572
C09937=1124.802,193.773,-64.448,-179.127,9.256,149.572
C09938=1124.799,194.022,-64.472,-179.125,9.259,149.572
C09939=1124.793,194.271,-64.497,-179.124,9.261,149.572
C09940=1124.789,194.519,-64.522,-179.122,9.264,149.572
C09941=1124.785,194.768,-64.547,-179.120,9.267,149.573
C09942=1124.780,195.017,-64.571,-179.118,9.269,149.573
C09943=1124.775,195.265,-64.595,-179.116,9.272,149.573
C09944=1124.771,195.514,-64.620,-179.114,9.274,149.573
C09945=1124.766,195.763,-64.645,-179.113,9.277,149.573
C09946=1124.762,196.011,-64.669,-179.111,9.280,149.573
C09947=1124.757,196.261,-64.694,-179.110,9.282,149.573
C09948=1124.753,196.509,-64.718,-179.106,9.286,149.573
C09949=1124.748,196.758,-64.742,-179.103,9.290,149.573
C09950=1124.744,197.007,-64.767,-179.099,9.293,149.573
C09951=1124.739,197.255,-64.792,-179.096,9.297,149.573
C09952=1124.735,197.504,-64.817,-179.092,9.300,149.573
C09953=1124.730,197.753,-64.841,-179.089,9.304,149.573
C09954=1124.726,198.002,-64.865,-179.085,9.308,149.573
C09955=1124.722,198.215,-64.887,-179.082,9.310,149.573
C09956=1124.719,198.429,-64.908,-179.079,9.314,149.573
C09957=1124.715,198.644,-64.929,-179.076,9.317,149.572
C09958=1124.710,198.858,-64.951,-179.073,9.320,149.572
C09959=1124.706,199.072,-64.972,-179.070,9.322,149.572
C09960=1124.703,199.286,-64.994,-179.067,9.325,149.572
C09961=1124.699,199.499,-65.015,-179.064,9.328,149.572
C09962=1124.695,199.714,-65.036,-179.062,9.331,149.572
C09963=1124.690,199.962,-65.061,-179.058,9.334,149.572
C09964=1124.686,200.211,-65.086,-179.055,9.338,149.572
C09965=1124.682,200.459,-65.111,-179.052,9.341,149.572
C09966=1124.677,200.709,-65.136,-179.048,9.344,149.571
C09967=1124.673,200.957,-65.160,-179.045,9.348,149.571
C09968=1124.669,201.206,-65.186,-179.042,9.350,149.571
C09969=1124.663,201.455,-65.211,-179.038,9.354,149.571
C09970=1124.660,201.703,-65.236,-179.035,9.357,149.571
C09971=1124.655,201.952,-65.261,-179.032,9.360,149.571
C09972=1124.651,202.201,-65.286,-179.029,9.363,149.571
C09973=1124.645,202.449,-65.311,-179.026,9.366,149.571
C09974=1124.642,202.698,-65.336,-179.023,9.370,149.571
C09975=1124.637,202.947,-65.361,-179.020,9.372,149.570
C09976=1124.633,203.196,-65.387,-179.017,9.375,149.570
C09977=1124.627,203.444,-65.411,-179.013,9.379,149.570
C09978=1124.624,203.693,-65.436,-179.010,9.381,149.570
C09979=1124.619,203.941,-65.461,-179.007,9.384,149.570
C09980=1124.615,204.190,-65.487,-179.005,9.387,149.570
C09981=1124.610,204.439,-65.513,-179.002,9.390,149.570
C09982=1124.605,204.688,-65.537,-178.999,9.393,149.570
C09983=1124.601,204.937,-65.563,-178.995,9.396,149.569
C09984=1124.596,205.185,-65.588,-178.993,9.399,149.570
C09985=1124.592,205.434,-65.613,-178.990,9.402,149.569
C09986=1124.588,205.682,-65.638,-178.987,9.405,149.569
C09987=1124.583,205.931,-65.664,-178.984,9.408,149.569
C09988=1124.579,206.180,-65.689,-178.981,9.411,149.569
C09989=1124.574,206.428,-65.714,-178.979,9.413,149.569
C09990=1124.570,206.677,-65.740,-178.976,9.416,149.569
C09991=1124.565,206.926,-65.765,-178.973,9.418,149.569
C09992=1124.560,207.175,-65.791,-178.970,9.421,149.569
C09993=1124.556,207.423,-65.816,-178.968,9.424,149.569
C09994=1124.551,207.671,-65.842,-178.965,9.427,149.569
C09995=1124.547,207.920,-65.867,-178.963,9.429,149.569
C09996=1124.543,208.169,-65.892,-178.960,9.432,149.569
//INST
///DATE 2021/06/15 17:28
///ATTR SC,RW,RJ
////FRAME ROBOT
///GROUP1 RB1
NOP
MOVL C00000 V=800.0 PL=0
MOVL C00001 V=800.0 PL=0
MOVL C00002 V=800.0 PL=0
MOVL C00003 V=800.0 PL=0
MOVL C00004 V=800.0 PL=0
MOVL C00005 V=800.0 PL=0
MOVL C00006 V=800.0 PL=0
MOVL C00007 V=800.0 PL=0
MOVL C00008 V=800.0 PL=0
MOVL C00009 V=800.0 PL=0
MOVL C00010 V=800.0 PL=0
MOVL C00011 V=800.0 PL=0
MOVL C00012 V=800.0 PL=0
MOVL C00013 V=800.0 PL=0
MOVL C00014 V=800.0 PL=0
MOVL C00015 V=800.0 PL=0
MOVL C00016 V=800.0 PL=0
MOVL C00017 V=800.0 PL=0
MOVL C00018 V=800.0 PL=0
MOVL C00019 V=800.0 PL=0
MOVL C00020 V=800.0 PL=0
MOVL C00021 V=800.0 PL=0
MOVL C00022 V=800.0 PL=0
MOVL C00023 V=800.0 PL=0
MOVL C00024 V=800.0 PL=0
MOVL C00025 V=800.0 PL=0
MOVL C00026 V=800.0 PL=0
MOVL C00027 V=800.0 PL=0
MOVL C00028 V=800.0 PL=0
MOVL C00029 V=800.0 PL=0
MOVL C00030 V=800.0 PL=0
MOVL C00031 V=800.0 PL=0
MOVL C00032 V=800.0 PL=0
MOVL C00033 V=800.0 PL=0
MOVL C00034 V=800.0 PL=0
MOVL C00035 V=800.0 PL=0
MOVL C00036 V=800.0 PL=0
MOVL C00037 V=800.0 PL=0
MOVL C00038 V=800.0 PL=0
MOVL C00039 V=800.0 PL=0
MOVL C00040 V=800.0 PL=0
MOVL C00041 V=800.0 PL=0
MOVL C00042 V=800.0 PL=0
MOVL C00043 V=800.0 PL=0
MOVL C00044 V=800.0 PL=0
MOVL C00045 V=800.0 PL=0
MOVL C00046 V=800.0 PL=0
MOVL C00047 V=800.0 PL=0
MOVL C00048 V=800.0 PL=0
MOVL C00049 V=800.0 PL=0
MOVL C00050 V=800.0 PL=0
MOVL C00051 V=800.0 PL=0
MOVL C00052 V=800.0 PL=0
MOVL C00053 V=800.0 PL=0
MOVL C00054 V=800.0 PL=0
MOVL C00055 V=800.0 PL=0
MOVL C00056 V=800.0 PL=0
MOVL C00057 V=800.0 PL=0
MOVL C00058 V=800.0 PL=0
MOVL C00059 V=800.0 PL=0
MOVL C00060 V=800.0 PL=0
MOVL C00061 V=800.0 PL=0
MOVL C00062 V=800.0 PL=0
MOVL C00063 V=800.0 PL=0
MOVL C00064 V=800.0 PL=0
MOVL C00065 V=800.0 PL=0
MOVL C00066 V=800.0 PL=0
MOVL C00067 V=800.0 PL=0
MOVL C00068 V=800.0 PL=0
MOVL C00069 V=800.0 PL=0
MOVL C00070 V=800.0 PL=0
MOVL C00071 V=800.0 PL=0
MOVL C00072 V=800.0 PL=0
MOVL C00073 V=800.0 PL=0
MOVL C00074 V=800.0 PL=0
MOVL C00075 V=800.0 PL=0
MOVL C00076 V=800.0 PL=0
MOVL C00077 V=800.0 PL=0
MOVL C00078 V=800.0 PL=0
MOVL C00079 V=800.0 PL=0
MOVL C00080 V=800.0 PL=0
MOVL C00081 V=800.0 PL=0
MOVL C00082 V=800.0 PL=0
MOVL C00083 V=800.0 PL=0
MOVL C00084 V=800.0 PL=0
MOVL C00085 V=800.0 PL=0
MOVL C00086 V=800.0 PL=0
MOVL C00087 V=800.0 PL=0
MOVL C00088 V=800.0 PL=0
MOVL C00089 V=800.0 PL=0
MOVL C00090 V=800.0 PL=0
MOVL C00091 V=800.0 PL=0
MOVL C00092 V=800.0 PL=0
MOVL C00093 V=800.0 PL=0
MOVL C00094 V=800.0 PL=0
MOVL C00095 V=800.0 PL=0
MOVL C00096 V=800.0 PL=0
MOVL C00097 V=800.0 PL=0
MOVL C00098 V=800.0 PL=0
MOVL C00099 V=800.0 PL=0
MOVL C00100 V=800.0 PL=0
MOVL C00101 V=800.0 PL=0
MOVL C00102 V=800.0 PL=0
MOVL C00103 V=800.0 PL=0
MOVL C00104 V=800.0 PL=0
MOVL C00105 V=800.0 PL=0
MOVL C00106 V=800.0 PL=0
MOVL C00107 V=800.0 PL=0
MOVL C00108 V=800.0 PL=0
MOVL C00109 V=800.0 PL=0
MOVL C00110 V=800.0 PL=0
MOVL C00111 V=800.0 PL=0
MOVL C00112 V=800.0 PL=0
MOVL C00113 V=800.0 PL=0
MOVL C00114 V=800.0 PL=0
MOVL C00115 V=800.0 PL=0
MOVL C00116 V=800.0 PL=0
MOVL C00117 V=800.0 PL=0
MOVL C00118 V=800.0 PL=0
MOVL C00119 V=800.0 PL=0
MOVL C00120 V=800.0 PL=0
MOVL C00121 V=800.0 PL=0
MOVL C00122 V=800.0 PL=0
MOVL C00123 V=800.0 PL=0
MOVL C00124 V=800.0 PL=0
MOVL C00125 V=800.0 PL=0
MOVL C00126 V=800.0 PL=0
MOVL C00127 V=800.0 PL=0
MOVL C00128 V=800.0 PL=0
MOVL C00129 V=800.0 PL=0
MOVL C00130 V=800.0 PL=0
MOVL C00131 V=800.0 PL=0
MOVL C00132 V=800.0 PL=0
MOVL C00133 V=800.0 PL=0
MOVL C00134 V=800.0 PL=0
MOVL C00135 V=800.0 PL=0
MOVL C00136 V=800.0 PL=0
MOVL C00137 V=800.0 PL=0
MOVL C00138 V=800.0 PL=0
MOVL C00139 V=800.0 PL=0
MOVL C00140 V=800.0 PL=0
MOVL C00141 V=800.0 PL=0
MOVL C00142 V=800.0 PL=0
MOVL C00143 V=800.0 PL=0
MOVL C00144 V=800.0 PL=0
MOVL C00145 V=800.0 PL=0
MOVL C00146 V=800.0 PL=0
MOVL C00147 V=800.0 PL=0
MOVL C00148 V=800.0 PL=0
MOVL C00149 V=800.0 PL=0
MOVL C00150 V=800.0 PL=0
MOVL C00151 V=800.0 PL=0
MOVL C00152 V=800.0 PL=0
MOVL C00153 V=800.0 PL=0
MOVL C00154 V=800.0 PL=0
MOVL C00155 V=800.0 PL=0
MOVL C00156 V=800.0 PL=0
MOVL C00157 V=800.0 PL=0
MOVL C00158 V=800.0 PL=0
MOVL C00159 V=800.0 PL=0
MOVL C00160 V=800.0 PL=0
MOVL C00161 V=800.0 PL=0
MOVL C00162 V=800.0 PL=0
MOVL C00163 V=800.0 PL=0
MOVL C00164 V=800.0 PL=0
MOVL C00165 V=800.0 PL=0
MOVL C00166 V=800.0 PL=0
MOVL C00167 V=800.0 PL=0
MOVL C00168 V=800.0 PL=0
MOVL C00169 V=800.0 PL=0
MOVL C00170 V=800.0 PL=0
MOVL C00171 V=800.0 PL=0
MOVL C00172 V=800.0 PL=0
MOVL C00173 V=800.0 PL=0
MOVL C00174 V=800.0 PL=0
MOVL C00175 V=800.0 PL=0
MOVL C00176 V=800.0 PL=0
MOVL C00177 V=800.0 PL=0
MOVL C00178 V=800.0 PL=0
MOVL C00179 V=800.0 PL=0
MOVL C00180 V=800.0 PL=0
MOVL C00181 V=800.0 PL=0
MOVL C00182 V=800.0 PL=0
MOVL C00183 V=800.0 PL=0
MOVL C00184 V=800.0 PL=0
MOVL C00185 V=800.0 PL=0
MOVL C00186 V=800.0 PL=0
MOVL C00187 V=800.0 PL=0
MOVL C00188 V=800.0 PL=0
MOVL C00189 V=800.0 PL=0
MOVL C00190 V=800.0 PL=0
MOVL C00191 V=800.0 PL=0
MOVL C00192 V=800.0 PL=0
MOVL C00193 V=800.0 PL=0
MOVL C00194 V=800.0 PL=0
MOVL C00195 V=800.0 PL=0
MOVL C00196 V=800.0 PL=0
MOVL C00197 V=800.0 PL=0
MOVL C00198 V=800.0 PL=0
MOVL C00199 V=800.0 PL=0
MOVL C00200 V=800.0 PL=0
MOVL C00201 V=800.0 PL=0
MOVL C00202 V=800.0 PL=0
MOVL C00203 V=800.0 PL=0
MOVL C00204 V=800.0 PL=0
MOVL C00205 V=800.0 PL=0
MOVL C00206 V=800.0 PL=0
MOVL C00207 V=800.0 PL=0
MOVL C00208 V=800.0 PL=0
MOVL C00209 V=800.0 PL=0
MOVL C00210 V=800.0 PL=0
MOVL C00211 V=800.0 PL=0
MOVL C00212 V=800.0 PL=0
MOVL C00213 V=800.0 PL=0
MOVL C00214 V=800.0 PL=0
MOVL C00215 V=800.0 PL=0
MOVL C00216 V=800.0 PL=0
MOVL C00217 V=800.0 PL=0
MOVL C00218 V=800.0 PL=0
MOVL C00219 V=800.0 PL=0
MOVL C00220 V=800.0 PL=0
MOVL C00221 V=800.0 PL=0
MOVL C00222 V=800.0 PL=0
MOVL C00223 V=800.0 PL=0
MOVL C00224 V=800.0 PL=0
MOVL C00225 V=800.0 PL=0
MOVL C00226 V=800.0 PL=0
MOVL C00227 V=800.0 PL=0
MOVL C00228 V=800.0 PL=0
MOVL C00229 V=800.0 PL=0
MOVL C00230 V=800.0 PL=0
MOVL C00231 V=800.0 PL=0
MOVL C00232 V=800.0 PL=0
MOVL C00233 V=800.0 PL=0
MOVL C00234 V=800.0 PL=0
MOVL C00235 V=800.0 PL=0
MOVL C00236 V=800.0 PL=0
MOVL C00237 V=800.0 PL=0
MOVL C00238 V=800.0 PL=0
MOVL C00239 V=800.0 PL=0
MOVL C00240 V=800.0 PL=0
MOVL C00241 V=800.0 PL=0
MOVL C00242 V=800.0 PL=0
MOVL C00243 V=800.0 PL=0
MOVL C00244 V=800.0 PL=0
MOVL C00245 V=800.0 PL=0
MOVL C00246 V=800.0 PL=0
MOVL C00247 V=800.0 PL=0
MOVL C00248 V=800.0 PL=0
MOVL C00249 V=800.0 PL=0
MOVL C00250 V=800.0 PL=0
MOVL C00251 V=800.0 PL=0
MOVL C00252 V=800.0 PL=0
MOVL C00253 V=800.0 PL=0
MOVL C00254 V=800.0 PL=0
MOVL C00255 V=800.0 PL=0
MOVL C00256 V=800.0 PL=0
MOVL C00257 V=800.0 PL=0
MOVL C00258 V=800.0 PL=0
MOVL C00259 V=800.0 PL=0
MOVL C00260 V=800.0 PL=0
MOVL C00261 V=800.0 PL=0
MOVL C00262 V=800.0 PL=0
MOVL C00263 V=800.0 PL=0
MOVL C00264 V=800.0 PL=0
MOVL C00265 V=800.0 PL=0
MOVL C00266 V=800.0 PL=0
MOVL C00267 V=800.0 PL=0
MOVL C00268 V=800.0 PL=0
MOVL C00269 V=800.0 PL=0
MOVL C00270 V=800.0 PL=0
MOVL C00271 V=800.0 PL=0
MOVL C00272 V=800.0 PL=0
MOVL C00273 V=800.0 PL=0
MOVL C00274 V=800.0 PL=0
MOVL C00275 V=800.0 PL=0
MOVL C00276 V=800.0 PL=0
MOVL C00277 V=800.0 PL=0
MOVL C00278 V=800.0 PL=0
MOVL C00279 V=800.0 PL=0
MOVL C00280 V=800.0 PL=0
MOVL C00281 V=800.0 PL=0
MOVL C00282 V=800.0 PL=0
MOVL C00283 V=800.0 PL=0
MOVL C00284 V=800.0 PL=0
MOVL C00285 V=800.0 PL=0
MOVL C00286 V=800.0 PL=0
MOVL C00287 V=800.0 PL=0
MOVL C00288 V=800.0 PL=0
MOVL C00289 V=800.0 PL=0
MOVL C00290 V=800.0 PL=0
MOVL C00291 V=800.0 PL=0
MOVL C00292 V=800.0 PL=0
MOVL C00293 V=800.0 PL=0
MOVL C00294 V=800.0 PL=0
MOVL C00295 V=800.0 PL=0
MOVL C00296 V=800.0 PL=0
MOVL C00297 V=800.0 PL=0
MOVL C00298 V=800.0 PL=0
MOVL C00299 V=800.0 PL=0
MOVL C00300 V=800.0 PL=0
MOVL C00301 V=800.0 PL=0
MOVL C00302 V=800.0 PL=0
MOVL C00303 V=800.0 PL=0
MOVL C00304 V=800.0 PL=0
MOVL C00305 V=800.0 PL=0
MOVL C00306 V=800.0 PL=0
MOVL C00307 V=800.0 PL=0
MOVL C00308 V=800.0 PL=0
MOVL C00309 V=800.0 PL=0
MOVL C00310 V=800.0 PL=0
MOVL C00311 V=800.0 PL=0
MOVL C00312 V=800.0 PL=0
MOVL C00313 V=800.0 PL=0
MOVL C00314 V=800.0 PL=0
MOVL C00315 V=800.0 PL=0
MOVL C00316 V=800.0 PL=0
MOVL C00317 V=800.0 PL=0
MOVL C00318 V=800.0 PL=0
MOVL C00319 V=800.0 PL=0
MOVL C00320 V=800.0 PL=0
MOVL C00321 V=800.0 PL=0
MOVL C00322 V=800.0 PL=0
MOVL C00323 V=800.0 PL=0
MOVL C00324 V=800.0 PL=0
MOVL C00325 V=800.0 PL=0
MOVL C00326 V=800.0 PL=0
MOVL C00327 V=800.0 PL=0
MOVL C00328 V=800.0 PL=0
MOVL C00329 V=800.0 PL=0
MOVL C00330 V=800.0 PL=0
MOVL C00331 V=800.0 PL=0
MOVL C00332 V=800.0 PL=0
MOVL C00333 V=800.0 PL=0
MOVL C00334 V=800.0 PL=0
MOVL C00335 V=800.0 PL=0
MOVL C00336 V=800.0 PL=0
MOVL C00337 V=800.0 PL=0
MOVL C00338 V=800.0 PL=0
MOVL C00339 V=800.0 PL=0
MOVL C00340 V=800.0 PL=0
MOVL C00341 V=800.0 PL=0
MOVL C00342 V=800.0 PL=0
MOVL C00343 V=800.0 PL=0
MOVL C00344 V=800.0 PL=0
MOVL C00345 V=800.0 PL=0
MOVL C00346 V=800.0 PL=0
MOVL C00347 V=800.0 PL=0
MOVL C00348 V=800.0 PL=0
MOVL C00349 V=800.0 PL=0
MOVL C00350 V=800.0 PL=0
MOVL C00351 V=800.0 PL=0
MOVL C00352 V=800.0 PL=0
MOVL C00353 V=800.0 PL=0
MOVL C00354 V=800.0 PL=0
MOVL C00355 V=800.0 PL=0
MOVL C00356 V=800.0 PL=0
MOVL C00357 V=800.0 PL=0
MOVL C00358 V=800.0 PL=0
MOVL C00359 V=800.0 PL=0
MOVL C00360 V=800.0 PL=0
MOVL C00361 V=800.0 PL=0
MOVL C00362 V=800.0 PL=0
MOVL C00363 V=800.0 PL=0
MOVL C00364 V=800.0 PL=0
MOVL C00365 V=800.0 PL=0
MOVL C00366 V=800.0 PL=0
MOVL C00367 V=800.0 PL=0
MOVL C00368 V=800.0 PL=0
MOVL C00369 V=800.0 PL=0
MOVL C00370 V=800.0 PL=0
MOVL C00371 V=800.0 PL=0
MOVL C00372 V=800.0 PL=0
MOVL C00373 V=800.0 PL=0
MOVL C00374 V=800.0 PL=0
MOVL C00375 V=800.0 PL=0
MOVL C00376 V=800.0 PL=0
MOVL C00377 V=800.0 PL=0
MOVL C00378 V=800.0 PL=0
MOVL C00379 V=800.0 PL=0
MOVL C00380 V=800.0 PL=0
MOVL C00381 V=800.0 PL=0
MOVL C00382 V=800.0 PL=0
MOVL C00383 V=800.0 PL=0
MOVL C00384 V=800.0 PL=0
MOVL C00385 V=800.0 PL=0
MOVL C00386 V=800.0 PL=0
MOVL C00387 V=800.0 PL=0
MOVL C00388 V=800.0 PL=0
MOVL C00389 V=800.0 PL=0
MOVL C00390 V=800.0 PL=0
MOVL C00391 V=800.0 PL=0
MOVL C00392 V=800.0 PL=0
MOVL C00393 V=800.0 PL=0
MOVL C00394 V=800.0 PL=0
MOVL C00395 V=800.0 PL=0
MOVL C00396 V=800.0 PL=0
MOVL C00397 V=800.0 PL=0
MOVL C00398 V=800.0 PL=0
MOVL C00399 V=800.0 PL=0
MOVL C00400 V=800.0 PL=0
MOVL C00401 V=800.0 PL=0
MOVL C00402 V=800.0 PL=0
MOVL C00403 V=800.0 PL=0
MOVL C00404 V=800.0 PL=0
MOVL C00405 V=800.0 PL=0
MOVL C00406 V=800.0 PL=0
MOVL C00407 V=800.0 PL=0
MOVL C00408 V=800.0 PL=0
MOVL C00409 V=800.0 PL=0
MOVL C00410 V=800.0 PL=0
MOVL C00411 V=800.0 PL=0
MOVL C00412 V=800.0 PL=0
MOVL C00413 V=800.0 PL=0
MOVL C00414 V=800.0 PL=0
MOVL C00415 V=800.0 PL=0
MOVL C00416 V=800.0 PL=0
MOVL C00417 V=800.0 PL=0
MOVL C00418 V=800.0 PL=0
MOVL C00419 V=800.0 PL=0
MOVL C00420 V=800.0 PL=0
MOVL C00421 V=800.0 PL=0
MOVL C00422 V=800.0 PL=0
MOVL C00423 V=800.0 PL=0
MOVL C00424 V=800.0 PL=0
MOVL C00425 V=800.0 PL=0
MOVL C00426 V=800.0 PL=0
MOVL C00427 V=800.0 PL=0
MOVL C00428 V=800.0 PL=0
MOVL C00429 V=800.0 PL=0
MOVL C00430 V=800.0 PL=0
MOVL C00431 V=800.0 PL=0
MOVL C00432 V=800.0 PL=0
MOVL C00433 V=800.0 PL=0
MOVL C00434 V=800.0 PL=0
MOVL C00435 V=800.0 PL=0
MOVL C00436 V=800.0 PL=0
MOVL C00437 V=800.0 PL=0
MOVL C00438 V=800.0 PL=0
MOVL C00439 V=800.0 PL=0
MOVL C00440 V=800.0 PL=0
MOVL C00441 V=800.0 PL=0
MOVL C00442 V=800.0 PL=0
MOVL C00443 V=800.0 PL=0
MOVL C00444 V=800.0 PL=0
MOVL C00445 V=800.0 PL=0
MOVL C00446 V=800.0 PL=0
MOVL C00447 V=800.0 PL=0
MOVL C00448 V=800.0 PL=0
MOVL C00449 V=800.0 PL=0
MOVL C00450 V=800.0 PL=0
MOVL C00451 V=800.0 PL=0
MOVL C00452 V=800.0 PL=0
MOVL C00453 V=800.0 PL=0
MOVL C00454 V=800.0 PL=0
MOVL C00455 V=800.0 PL=0
MOVL C00456 V=800.0 PL=0
MOVL C00457 V=800.0 PL=0
MOVL C00458 V=800.0 PL=0
MOVL C00459 V=800.0 PL=0
MOVL C00460 V=800.0 PL=0
MOVL C00461 V=800.0 PL=0
MOVL C00462 V=800.0 PL=0
MOVL C00463 V=800.0 PL=0
MOVL C00464 V=800.0 PL=0
MOVL C00465 V=800.0 PL=0
MOVL C00466 V=800.0 PL=0
MOVL C00467 V=800.0 PL=0
MOVL C00468 V=800.0 PL=0
MOVL C00469 V=800.0 PL=0
MOVL C00470 V=800.0 PL=0
MOVL C00471 V=800.0 PL=0
MOVL C00472 V=800.0 PL=0
MOVL C00473 V=800.0 PL=0
MOVL C00474 V=800.0 PL=0
MOVL C00475 V=800.0 PL=0
MOVL C00476 V=800.0 PL=0
MOVL C00477 V=800.0 PL=0
MOVL C00478 V=800.0 PL=0
MOVL C00479 V=800.0 PL=0
MOVL C00480 V=800.0 PL=0
MOVL C00481 V=800.0 PL=0
MOVL C00482 V=800.0 PL=0
MOVL C00483 V=800.0 PL=0
MOVL C00484 V=800.0 PL=0
MOVL C00485 V=800.0 PL=0
MOVL C00486 V=800.0 PL=0
MOVL C00487 V=800.0 PL=0
MOVL C00488 V=800.0 PL=0
MOVL C00489 V=800.0 PL=0
MOVL C00490 V=800.0 PL=0
MOVL C00491 V=800.0 PL=0
MOVL C00492 V=800.0 PL=0
MOVL C00493 V=800.0 PL=0
MOVL C00494 V=800.0 PL=0
MOVL C00495 V=800.0 PL=0
MOVL C00496 V=800.0 PL=0
MOVL C00497 V=800.0 PL=0
MOVL C00498 V=800.0 PL=0
MOVL C00499 V=800.0 PL=0
MOVL C00500 V=800.0 PL=0
MOVL C00501 V=800.0 PL=0
MOVL C00502 V=800.0 PL=0
MOVL C00503 V=800.0 PL=0
MOVL C00504 V=800.0 PL=0
MOVL C00505 V=800.0 PL=0
MOVL C00506 V=800.0 PL=0
MOVL C00507 V=800.0 PL=0
MOVL C00508 V=800.0 PL=0
MOVL C00509 V=800.0 PL=0
MOVL C00510 V=800.0 PL=0
MOVL C00511 V=800.0 PL=0
MOVL C00512 V=800.0 PL=0
MOVL C00513 V=800.0 PL=0
MOVL C00514 V=800.0 PL=0
MOVL C00515 V=800.0 PL=0
MOVL C00516 V=800.0 PL=0
MOVL C00517 V=800.0 PL=0
MOVL C00518 V=800.0 PL=0
MOVL C00519 V=800.0 PL=0
MOVL C00520 V=800.0 PL=0
MOVL C00521 V=800.0 PL=0
MOVL C00522 V=800.0 PL=0
MOVL C00523 V=800.0 PL=0
MOVL C00524 V=800.0 PL=0
MOVL C00525 V=800.0 PL=0
MOVL C00526 V=800.0 PL=0
MOVL C00527 V=800.0 PL=0
MOVL C00528 V=800.0 PL=0
MOVL C00529 V=800.0 PL=0
MOVL C00530 V=800.0 PL=0
MOVL C00531 V=800.0 PL=0
MOVL C00532 V=800.0 PL=0
MOVL C00533 V=800.0 PL=0
MOVL C00534 V=800.0 PL=0
MOVL C00535 V=800.0 PL=0
MOVL C00536 V=800.0 PL=0
MOVL C00537 V=800.0 PL=0
MOVL C00538 V=800.0 PL=0
MOVL C00539 V=800.0 PL=0
MOVL C00540 V=800.0 PL=0
MOVL C00541 V=800.0 PL=0
MOVL C00542 V=800.0 PL=0
MOVL C00543 V=800.0 PL=0
MOVL C00544 V=800.0 PL=0
MOVL C00545 V=800.0 PL=0
MOVL C00546 V=800.0 PL=0
MOVL C00547 V=800.0 PL=0
MOVL C00548 V=800.0 PL=0
MOVL C00549 V=800.0 PL=0
MOVL C00550 V=800.0 PL=0
MOVL C00551 V=800.0 PL=0
MOVL C00552 V=800.0 PL=0
MOVL C00553 V=800.0 PL=0
MOVL C00554 V=800.0 PL=0
MOVL C00555 V=800.0 PL=0
MOVL C00556 V=800.0 PL=0
MOVL C00557 V=800.0 PL=0
MOVL C00558 V=800.0 PL=0
MOVL C00559 V=800.0 PL=0
MOVL C00560 V=800.0 PL=0
MOVL C00561 V=800.0 PL=0
MOVL C00562 V=800.0 PL=0
MOVL C00563 V=800.0 PL=0
MOVL C00564 V=800.0 PL=0
MOVL C00565 V=800.0 PL=0
MOVL C00566 V=800.0 PL=0
MOVL C00567 V=800.0 PL=0
MOVL C00568 V=800.0 PL=0
MOVL C00569 V=800.0 PL=0
MOVL C00570 V=800.0 PL=0
MOVL C00571 V=800.0 PL=0
MOVL C00572 V=800.0 PL=0
MOVL C00573 V=800.0 PL=0
MOVL C00574 V=800.0 PL=0
MOVL C00575 V=800.0 PL=0
MOVL C00576 V=800.0 PL=0
MOVL C00577 V=800.0 PL=0
MOVL C00578 V=800.0 PL=0
MOVL C00579 V=800.0 PL=0
MOVL C00580 V=800.0 PL=0
MOVL C00581 V=800.0 PL=0
MOVL C00582 V=800.0 PL=0
MOVL C00583 V=800.0 PL=0
MOVL C00584 V=800.0 PL=0
MOVL C00585 V=800.0 PL=0
MOVL C00586 V=800.0 PL=0
MOVL C00587 V=800.0 PL=0
MOVL C00588 V=800.0 PL=0
MOVL C00589 V=800.0 PL=0
MOVL C00590 V=800.0 PL=0
MOVL C00591 V=800.0 PL=0
MOVL C00592 V=800.0 PL=0
MOVL C00593 V=800.0 PL=0
MOVL C00594 V=800.0 PL=0
MOVL C00595 V=800.0 PL=0
MOVL C00596 V=800.0 PL=0
MOVL C00597 V=800.0 PL=0
MOVL C00598 V=800.0 PL=0
MOVL C00599 V=800.0 PL=0
MOVL C00600 V=800.0 PL=0
MOVL C00601 V=800.0 PL=0
MOVL C00602 V=800.0 PL=0
MOVL C00603 V=800.0 PL=0
MOVL C00604 V=800.0 PL=0
MOVL C00605 V=800.0 PL=0
MOVL C00606 V=800.0 PL=0
MOVL C00607 V=800.0 PL=0
MOVL C00608 V=800.0 PL=0
MOVL C00609 V=800.0 PL=0
MOVL C00610 V=800.0 PL=0
MOVL C00611 V=800.0 PL=0
MOVL C00612 V=800.0 PL=0
MOVL C00613 V=800.0 PL=0
MOVL C00614 V=800.0 PL=0
MOVL C00615 V=800.0 PL=0
MOVL C00616 V=800.0 PL=0
MOVL C00617 V=800.0 PL=0
MOVL C00618 V=800.0 PL=0
MOVL C00619 V=800.0 PL=0
MOVL C00620 V=800.0 PL=0
MOVL C00621 V=800.0 PL=0
MOVL C00622 V=800.0 PL=0
MOVL C00623 V=800.0 PL=0
MOVL C00624 V=800.0 PL=0
MOVL C00625 V=800.0 PL=0
MOVL C00626 V=800.0 PL=0
MOVL C00627 V=800.0 PL=0
MOVL C00628 V=800.0 PL=0
MOVL C00629 V=800.0 PL=0
MOVL C00630 V=800.0 PL=0
MOVL C00631 V=800.0 PL=0
MOVL C00632 V=800.0 PL=0
MOVL C00633 V=800.0 PL=0
MOVL C00634 V=800.0 PL=0
MOVL C00635 V=800.0 PL=0
MOVL C00636 V=800.0 PL=0
MOVL C00637 V=800.0 PL=0
MOVL C00638 V=800.0 PL=0
MOVL C00639 V=800.0 PL=0
MOVL C00640 V=800.0 PL=0
MOVL C00641 V=800.0 PL=0
MOVL C00642 V=800.0 PL=0
MOVL C00643 V=800.0 PL=0
MOVL C00644 V=800.0 PL=0
MOVL C00645 V=800.0 PL=0
MOVL C00646 V=800.0 PL=0
MOVL C00647 V=800.0 PL=0
MOVL C00648 V=800.0 PL=0
MOVL C00649 V=800.0 PL=0
MOVL C00650 V=800.0 PL=0
MOVL C00651 V=800.0 PL=0
MOVL C00652 V=800.0 PL=0
MOVL C00653 V=800.0 PL=0
MOVL C00654 V=800.0 PL=0
MOVL C00655 V=800.0 PL=0
MOVL C00656 V=800.0 PL=0
MOVL C00657 V=800.0 PL=0
MOVL C00658 V=800.0 PL=0
MOVL C00659 V=800.0 PL=0
MOVL C00660 V=800.0 PL=0
MOVL C00661 V=800.0 PL=0
MOVL C00662 V=800.0 PL=0
MOVL C00663 V=800.0 PL=0
MOVL C00664 V=800.0 PL=0
MOVL C00665 V=800.0 PL=0
MOVL C00666 V=800.0 PL=0
MOVL C00667 V=800.0 PL=0
MOVL C00668 V=800.0 PL=0
MOVL C00669 V=800.0 PL=0
MOVL C00670 V=800.0 PL=0
MOVL C00671 V=800.0 PL=0
MOVL C00672 V=800.0 PL=0
MOVL C00673 V=800.0 PL=0
MOVL C00674 V=800.0 PL=0
MOVL C00675 V=800.0 PL=0
MOVL C00676 V=800.0 PL=0
MOVL C00677 V=800.0 PL=0
MOVL C00678 V=800.0 PL=0
MOVL C00679 V=800.0 PL=0
MOVL C00680 V=800.0 PL=0
MOVL C00681 V=800.0 PL=0
MOVL C00682 V=800.0 PL=0
MOVL C00683 V=800.0 PL=0
MOVL C00684 V=800.0 PL=0
MOVL C00685 V=800.0 PL=0
MOVL C00686 V=800.0 PL=0
MOVL C00687 V=800.0 PL=0
MOVL C00688 V=800.0 PL=0
MOVL C00689 V=800.0 PL=0
MOVL C00690 V=800.0 PL=0
MOVL C00691 V=800.0 PL=0
MOVL C00692 V=800.0 PL=0
MOVL C00693 V=800.0 PL=0
MOVL C00694 V=800.0 PL=0
MOVL C00695 V=800.0 PL=0
MOVL C00696 V=800.0 PL=0
MOVL C00697 V=800.0 PL=0
MOVL C00698 V=800.0 PL=0
MOVL C00699 V=800.0 PL=0
MOVL C00700 V=800.0 PL=0
MOVL C00701 V=800.0 PL=0
MOVL C00702 V=800.0 PL=0
MOVL C00703 V=800.0 PL=0
MOVL C00704 V=800.0 PL=0
MOVL C00705 V=800.0 PL=0
MOVL C00706 V=800.0 PL=0
MOVL C00707 V=800.0 PL=0
MOVL C00708 V=800.0 PL=0
MOVL C00709 V=800.0 PL=0
MOVL C00710 V=800.0 PL=0
MOVL C00711 V=800.0 PL=0
MOVL C00712 V=800.0 PL=0
MOVL C00713 V=800.0 PL=0
MOVL C00714 V=800.0 PL=0
MOVL C00715 V=800.0 PL=0
MOVL C00716 V=800.0 PL=0
MOVL C00717 V=800.0 PL=0
MOVL C00718 V=800.0 PL=0
MOVL C00719 V=800.0 PL=0
MOVL C00720 V=800.0 PL=0
MOVL C00721 V=800.0 PL=0
MOVL C00722 V=800.0 PL=0
MOVL C00723 V=800.0 PL=0
MOVL C00724 V=800.0 PL=0
MOVL C00725 V=800.0 PL=0
MOVL C00726 V=800.0 PL=0
MOVL C00727 V=800.0 PL=0
MOVL C00728 V=800.0 PL=0
MOVL C00729 V=800.0 PL=0
MOVL C00730 V=800.0 PL=0
MOVL C00731 V=800.0 PL=0
MOVL C00732 V=800.0 PL=0
MOVL C00733 V=800.0 PL=0
MOVL C00734 V=800.0 PL=0
MOVL C00735 V=800.0 PL=0
MOVL C00736 V=800.0 PL=0
MOVL C00737 V=800.0 PL=0
MOVL C00738 V=800.0 PL=0
MOVL C00739 V=800.0 PL=0
MOVL C00740 V=800.0 PL=0
MOVL C00741 V=800.0 PL=0
MOVL C00742 V=800.0 PL=0
MOVL C00743 V=800.0 PL=0
MOVL C00744 V=800.0 PL=0
MOVL C00745 V=800.0 PL=0
MOVL C00746 V=800.0 PL=0
MOVL C00747 V=800.0 PL=0
MOVL C00748 V=800.0 PL=0
MOVL C00749 V=800.0 PL=0
MOVL C00750 V=800.0 PL=0
MOVL C00751 V=800.0 PL=0
MOVL C00752 V=800.0 PL=0
MOVL C00753 V=800.0 PL=0
MOVL C00754 V=800.0 PL=0
MOVL C00755 V=800.0 PL=0
MOVL C00756 V=800.0 PL=0
MOVL C00757 V=800.0 PL=0
MOVL C00758 V=800.0 PL=0
MOVL C00759 V=800.0 PL=0
MOVL C00760 V=800.0 PL=0
MOVL C00761 V=800.0 PL=0
MOVL C00762 V=800.0 PL=0
MOVL C00763 V=800.0 PL=0
MOVL C00764 V=800.0 PL=0
MOVL C00765 V=800.0 PL=0
MOVL C00766 V=800.0 PL=0
MOVL C00767 V=800.0 PL=0
MOVL C00768 V=800.0 PL=0
MOVL C00769 V=800.0 PL=0
MOVL C00770 V=800.0 PL=0
MOVL C00771 V=800.0 PL=0
MOVL C00772 V=800.0 PL=0
MOVL C00773 V=800.0 PL=0
MOVL C00774 V=800.0 PL=0
MOVL C00775 V=800.0 PL=0
MOVL C00776 V=800.0 PL=0
MOVL C00777 V=800.0 PL=0
MOVL C00778 V=800.0 PL=0
MOVL C00779 V=800.0 PL=0
MOVL C00780 V=800.0 PL=0
MOVL C00781 V=800.0 PL=0
MOVL C00782 V=800.0 PL=0
MOVL C00783 V=800.0 PL=0
MOVL C00784 V=800.0 PL=0
MOVL C00785 V=800.0 PL=0
MOVL C00786 V=800.0 PL=0
MOVL C00787 V=800.0 PL=0
MOVL C00788 V=800.0 PL=0
MOVL C00789 V=800.0 PL=0
MOVL C00790 V=800.0 PL=0
MOVL C00791 V=800.0 PL=0
MOVL C00792 V=800.0 PL=0
MOVL C00793 V=800.0 PL=0
MOVL C00794 V=800.0 PL=0
MOVL C00795 V=800.0 PL=0
MOVL C00796 V=800.0 PL=0
MOVL C00797 V=800.0 PL=0
MOVL C00798 V=800.0 PL=0
MOVL C00799 V=800.0 PL=0
MOVL C00800 V=800.0 PL=0
MOVL C00801 V=800.0 PL=0
MOVL C00802 V=800.0 PL=0
MOVL C00803 V=800.0 PL=0
MOVL C00804 V=800.0 PL=0
MOVL C00805 V=800.0 PL=0
MOVL C00806 V=800.0 PL=0
MOVL C00807 V=800.0 PL=0
MOVL C00808 V=800.0 PL=0
MOVL C00809 V=800.0 PL=0
MOVL C00810 V=800.0 PL=0
MOVL C00811 V=800.0 PL=0
MOVL C00812 V=800.0 PL=0
MOVL C00813 V=800.0 PL=0
MOVL C00814 V=800.0 PL=0
MOVL C00815 V=800.0 PL=0
MOVL C00816 V=800.0 PL=0
MOVL C00817 V=800.0 PL=0
MOVL C00818 V=800.0 PL=0
MOVL C00819 V=800.0 PL=0
MOVL C00820 V=800.0 PL=0
MOVL C00821 V=800.0 PL=0
MOVL C00822 V=800.0 PL=0
MOVL C00823 V=800.0 PL=0
MOVL C00824 V=800.0 PL=0
MOVL C00825 V=800.0 PL=0
MOVL C00826 V=800.0 PL=0
MOVL C00827 V=800.0 PL=0
MOVL C00828 V=800.0 PL=0
MOVL C00829 V=800.0 PL=0
MOVL C00830 V=800.0 PL=0
MOVL C00831 V=800.0 PL=0
MOVL C00832 V=800.0 PL=0
MOVL C00833 V=800.0 PL=0
MOVL C00834 V=800.0 PL=0
MOVL C00835 V=800.0 PL=0
MOVL C00836 V=800.0 PL=0
MOVL C00837 V=800.0 PL=0
MOVL C00838 V=800.0 PL=0
MOVL C00839 V=800.0 PL=0
MOVL C00840 V=800.0 PL=0
MOVL C00841 V=800.0 PL=0
MOVL C00842 V=800.0 PL=0
MOVL C00843 V=800.0 PL=0
MOVL C00844 V=800.0 PL=0
MOVL C00845 V=800.0 PL=0
MOVL C00846 V=800.0 PL=0
MOVL C00847 V=800.0 PL=0
MOVL C00848 V=800.0 PL=0
MOVL C00849 V=800.0 PL=0
MOVL C00850 V=800.0 PL=0
MOVL C00851 V=800.0 PL=0
MOVL C00852 V=800.0 PL=0
MOVL C00853 V=800.0 PL=0
MOVL C00854 V=800.0 PL=0
MOVL C00855 V=800.0 PL=0
MOVL C00856 V=800.0 PL=0
MOVL C00857 V=800.0 PL=0
MOVL C00858 V=800.0 PL=0
MOVL C00859 V=800.0 PL=0
MOVL C00860 V=800.0 PL=0
MOVL C00861 V=800.0 PL=0
MOVL C00862 V=800.0 PL=0
MOVL C00863 V=800.0 PL=0
MOVL C00864 V=800.0 PL=0
MOVL C00865 V=800.0 PL=0
MOVL C00866 V=800.0 PL=0
MOVL C00867 V=800.0 PL=0
MOVL C00868 V=800.0 PL=0
MOVL C00869 V=800.0 PL=0
MOVL C00870 V=800.0 PL=0
MOVL C00871 V=800.0 PL=0
MOVL C00872 V=800.0 PL=0
MOVL C00873 V=800.0 PL=0
MOVL C00874 V=800.0 PL=0
MOVL C00875 V=800.0 PL=0
MOVL C00876 V=800.0 PL=0
MOVL C00877 V=800.0 PL=0
MOVL C00878 V=800.0 PL=0
MOVL C00879 V=800.0 PL=0
MOVL C00880 V=800.0 PL=0
MOVL C00881 V=800.0 PL=0
MOVL C00882 V=800.0 PL=0
MOVL C00883 V=800.0 PL=0
MOVL C00884 V=800.0 PL=0
MOVL C00885 V=800.0 PL=0
MOVL C00886 V=800.0 PL=0
MOVL C00887 V=800.0 PL=0
MOVL C00888 V=800.0 PL=0
MOVL C00889 V=800.0 PL=0
MOVL C00890 V=800.0 PL=0
MOVL C00891 V=800.0 PL=0
MOVL C00892 V=800.0 PL=0
MOVL C00893 V=800.0 PL=0
MOVL C00894 V=800.0 PL=0
MOVL C00895 V=800.0 PL=0
MOVL C00896 V=800.0 PL=0
MOVL C00897 V=800.0 PL=0
MOVL C00898 V=800.0 PL=0
MOVL C00899 V=800.0 PL=0
MOVL C00900 V=800.0 PL=0
MOVL C00901 V=800.0 PL=0
MOVL C00902 V=800.0 PL=0
MOVL C00903 V=800.0 PL=0
MOVL C00904 V=800.0 PL=0
MOVL C00905 V=800.0 PL=0
MOVL C00906 V=800.0 PL=0
MOVL C00907 V=800.0 PL=0
MOVL C00908 V=800.0 PL=0
MOVL C00909 V=800.0 PL=0
MOVL C00910 V=800.0 PL=0
MOVL C00911 V=800.0 PL=0
MOVL C00912 V=800.0 PL=0
MOVL C00913 V=800.0 PL=0
MOVL C00914 V=800.0 PL=0
MOVL C00915 V=800.0 PL=0
MOVL C00916 V=800.0 PL=0
MOVL C00917 V=800.0 PL=0
MOVL C00918 V=800.0 PL=0
MOVL C00919 V=800.0 PL=0
MOVL C00920 V=800.0 PL=0
MOVL C00921 V=800.0 PL=0
MOVL C00922 V=800.0 PL=0
MOVL C00923 V=800.0 PL=0
MOVL C00924 V=800.0 PL=0
MOVL C00925 V=800.0 PL=0
MOVL C00926 V=800.0 PL=0
MOVL C00927 V=800.0 PL=0
MOVL C00928 V=800.0 PL=0
MOVL C00929 V=800.0 PL=0
MOVL C00930 V=800.0 PL=0
MOVL C00931 V=800.0 PL=0
MOVL C00932 V=800.0 PL=0
MOVL C00933 V=800.0 PL=0
MOVL C00934 V=800.0 PL=0
MOVL C00935 V=800.0 PL=0
MOVL C00936 V=800.0 PL=0
MOVL C00937 V=800.0 PL=0
MOVL C00938 V=800.0 PL=0
MOVL C00939 V=800.0 PL=0
MOVL C00940 V=800.0 PL=0
MOVL C00941 V=800.0 PL=0
MOVL C00942 V=800.0 PL=0
MOVL C00943 V=800.0 PL=0
MOVL C00944 V=800.0 PL=0
MOVL C00945 V=800.0 PL=0
MOVL C00946 V=800.0 PL=0
MOVL C00947 V=800.0 PL=0
MOVL C00948 V=800.0 PL=0
MOVL C00949 V=800.0 PL=0
MOVL C00950 V=800.0 PL=0
MOVL C00951 V=800.0 PL=0
MOVL C00952 V=800.0 PL=0
MOVL C00953 V=800.0 PL=0
MOVL C00954 V=800.0 PL=0
MOVL C00955 V=800.0 PL=0
MOVL C00956 V=800.0 PL=0
MOVL C00957 V=800.0 PL=0
MOVL C00958 V=800.0 PL=0
MOVL C00959 V=800.0 PL=0
MOVL C00960 V=800.0 PL=0
MOVL C00961 V=800.0 PL=0
MOVL C00962 V=800.0 PL=0
MOVL C00963 V=800.0 PL=0
MOVL C00964 V=800.0 PL=0
MOVL C00965 V=800.0 PL=0
MOVL C00966 V=800.0 PL=0
MOVL C00967 V=800.0 PL=0
MOVL C00968 V=800.0 PL=0
MOVL C00969 V=800.0 PL=0
MOVL C00970 V=800.0 PL=0
MOVL C00971 V=800.0 PL=0
MOVL C00972 V=800.0 PL=0
MOVL C00973 V=800.0 PL=0
MOVL C00974 V=800.0 PL=0
MOVL C00975 V=800.0 PL=0
MOVL C00976 V=800.0 PL=0
MOVL C00977 V=800.0 PL=0
MOVL C00978 V=800.0 PL=0
MOVL C00979 V=800.0 PL=0
MOVL C00980 V=800.0 PL=0
MOVL C00981 V=800.0 PL=0
MOVL C00982 V=800.0 PL=0
MOVL C00983 V=800.0 PL=0
MOVL C00984 V=800.0 PL=0
MOVL C00985 V=800.0 PL=0
MOVL C00986 V=800.0 PL=0
MOVL C00987 V=800.0 PL=0
MOVL C00988 V=800.0 PL=0
MOVL C00989 V=800.0 PL=0
MOVL C00990 V=800.0 PL=0
MOVL C00991 V=800.0 PL=0
MOVL C00992 V=800.0 PL=0
MOVL C00993 V=800.0 PL=0
MOVL C00994 V=800.0 PL=0
MOVL C00995 V=800.0 PL=0
MOVL C00996 V=800.0 PL=0
MOVL C00997 V=800.0 PL=0
MOVL C00998 V=800.0 PL=0
MOVL C00999 V=800.0 PL=0
MOVL C01000 V=800.0 PL=0
MOVL C01001 V=800.0 PL=0
MOVL C01002 V=800.0 PL=0
MOVL C01003 V=800.0 PL=0
MOVL C01004 V=800.0 PL=0
MOVL C01005 V=800.0 PL=0
MOVL C01006 V=800.0 PL=0
MOVL C01007 V=800.0 PL=0
MOVL C01008 V=800.0 PL=0
MOVL C01009 V=800.0 PL=0
MOVL C01010 V=800.0 PL=0
MOVL C01011 V=800.0 PL=0
MOVL C01012 V=800.0 PL=0
MOVL C01013 V=800.0 PL=0
MOVL C01014 V=800.0 PL=0
MOVL C01015 V=800.0 PL=0
MOVL C01016 V=800.0 PL=0
MOVL C01017 V=800.0 PL=0
MOVL C01018 V=800.0 PL=0
MOVL C01019 V=800.0 PL=0
MOVL C01020 V=800.0 PL=0
MOVL C01021 V=800.0 PL=0
MOVL C01022 V=800.0 PL=0
MOVL C01023 V=800.0 PL=0
MOVL C01024 V=800.0 PL=0
MOVL C01025 V=800.0 PL=0
MOVL C01026 V=800.0 PL=0
MOVL C01027 V=800.0 PL=0
MOVL C01028 V=800.0 PL=0
MOVL C01029 V=800.0 PL=0
MOVL C01030 V=800.0 PL=0
MOVL C01031 V=800.0 PL=0
MOVL C01032 V=800.0 PL=0
MOVL C01033 V=800.0 PL=0
MOVL C01034 V=800.0 PL=0
MOVL C01035 V=800.0 PL=0
MOVL C01036 V=800.0 PL=0
MOVL C01037 V=800.0 PL=0
MOVL C01038 V=800.0 PL=0
MOVL C01039 V=800.0 PL=0
MOVL C01040 V=800.0 PL=0
MOVL C01041 V=800.0 PL=0
MOVL C01042 V=800.0 PL=0
MOVL C01043 V=800.0 PL=0
MOVL C01044 V=800.0 PL=0
MOVL C01045 V=800.0 PL=0
MOVL C01046 V=800.0 PL=0
MOVL C01047 V=800.0 PL=0
MOVL C01048 V=800.0 PL=0
MOVL C01049 V=800.0 PL=0
MOVL C01050 V=800.0 PL=0
MOVL C01051 V=800.0 PL=0
MOVL C01052 V=800.0 PL=0
MOVL C01053 V=800.0 PL=0
MOVL C01054 V=800.0 PL=0
MOVL C01055 V=800.0 PL=0
MOVL C01056 V=800.0 PL=0
MOVL C01057 V=800.0 PL=0
MOVL C01058 V=800.0 PL=0
MOVL C01059 V=800.0 PL=0
MOVL C01060 V=800.0 PL=0
MOVL C01061 V=800.0 PL=0
MOVL C01062 V=800.0 PL=0
MOVL C01063 V=800.0 PL=0
MOVL C01064 V=800.0 PL=0
MOVL C01065 V=800.0 PL=0
MOVL C01066 V=800.0 PL=0
MOVL C01067 V=800.0 PL=0
MOVL C01068 V=800.0 PL=0
MOVL C01069 V=800.0 PL=0
MOVL C01070 V=800.0 PL=0
MOVL C01071 V=800.0 PL=0
MOVL C01072 V=800.0 PL=0
MOVL C01073 V=800.0 PL=0
MOVL C01074 V=800.0 PL=0
MOVL C01075 V=800.0 PL=0
MOVL C01076 V=800.0 PL=0
MOVL C01077 V=800.0 PL=0
MOVL C01078 V=800.0 PL=0
MOVL C01079 V=800.0 PL=0
MOVL C01080 V=800.0 PL=0
MOVL C01081 V=800.0 PL=0
MOVL C01082 V=800.0 PL=0
MOVL C01083 V=800.0 PL=0
MOVL C01084 V=800.0 PL=0
MOVL C01085 V=800.0 PL=0
MOVL C01086 V=800.0 PL=0
MOVL C01087 V=800.0 PL=0
MOVL C01088 V=800.0 PL=0
MOVL C01089 V=800.0 PL=0
MOVL C01090 V=800.0 PL=0
MOVL C01091 V=800.0 PL=0
MOVL C01092 V=800.0 PL=0
MOVL C01093 V=800.0 PL=0
MOVL C01094 V=800.0 PL=0
MOVL C01095 V=800.0 PL=0
MOVL C01096 V=800.0 PL=0
MOVL C01097 V=800.0 PL=0
MOVL C01098 V=800.0 PL=0
MOVL C01099 V=800.0 PL=0
MOVL C01100 V=800.0 PL=0
MOVL C01101 V=800.0 PL=0
MOVL C01102 V=800.0 PL=0
MOVL C01103 V=800.0 PL=0
MOVL C01104 V=800.0 PL=0
MOVL C01105 V=800.0 PL=0
MOVL C01106 V=800.0 PL=0
MOVL C01107 V=800.0 PL=0
MOVL C01108 V=800.0 PL=0
MOVL C01109 V=800.0 PL=0
MOVL C01110 V=800.0 PL=0
MOVL C01111 V=800.0 PL=0
MOVL C01112 V=800.0 PL=0
MOVL C01113 V=800.0 PL=0
MOVL C01114 V=800.0 PL=0
MOVL C01115 V=800.0 PL=0
MOVL C01116 V=800.0 PL=0
MOVL C01117 V=800.0 PL=0
MOVL C01118 V=800.0 PL=0
MOVL C01119 V=800.0 PL=0
MOVL C01120 V=800.0 PL=0
MOVL C01121 V=800.0 PL=0
MOVL C01122 V=800.0 PL=0
MOVL C01123 V=800.0 PL=0
MOVL C01124 V=800.0 PL=0
MOVL C01125 V=800.0 PL=0
MOVL C01126 V=800.0 PL=0
MOVL C01127 V=800.0 PL=0
MOVL C01128 V=800.0 PL=0
MOVL C01129 V=800.0 PL=0
MOVL C01130 V=800.0 PL=0
MOVL C01131 V=800.0 PL=0
MOVL C01132 V=800.0 PL=0
MOVL C01133 V=800.0 PL=0
MOVL C01134 V=800.0 PL=0
MOVL C01135 V=800.0 PL=0
MOVL C01136 V=800.0 PL=0
MOVL C01137 V=800.0 PL=0
MOVL C01138 V=800.0 PL=0
MOVL C01139 V=800.0 PL=0
MOVL C01140 V=800.0 PL=0
MOVL C01141 V=800.0 PL=0
MOVL C01142 V=800.0 PL=0
MOVL C01143 V=800.0 PL=0
MOVL C01144 V=800.0 PL=0
MOVL C01145 V=800.0 PL=0
MOVL C01146 V=800.0 PL=0
MOVL C01147 V=800.0 PL=0
MOVL C01148 V=800.0 PL=0
MOVL C01149 V=800.0 PL=0
MOVL C01150 V=800.0 PL=0
MOVL C01151 V=800.0 PL=0
MOVL C01152 V=800.0 PL=0
MOVL C01153 V=800.0 PL=0
MOVL C01154 V=800.0 PL=0
MOVL C01155 V=800.0 PL=0
MOVL C01156 V=800.0 PL=0
MOVL C01157 V=800.0 PL=0
MOVL C01158 V=800.0 PL=0
MOVL C01159 V=800.0 PL=0
MOVL C01160 V=800.0 PL=0
MOVL C01161 V=800.0 PL=0
MOVL C01162 V=800.0 PL=0
MOVL C01163 V=800.0 PL=0
MOVL C01164 V=800.0 PL=0
MOVL C01165 V=800.0 PL=0
MOVL C01166 V=800.0 PL=0
MOVL C01167 V=800.0 PL=0
MOVL C01168 V=800.0 PL=0
MOVL C01169 V=800.0 PL=0
MOVL C01170 V=800.0 PL=0
MOVL C01171 V=800.0 PL=0
MOVL C01172 V=800.0 PL=0
MOVL C01173 V=800.0 PL=0
MOVL C01174 V=800.0 PL=0
MOVL C01175 V=800.0 PL=0
MOVL C01176 V=800.0 PL=0
MOVL C01177 V=800.0 PL=0
MOVL C01178 V=800.0 PL=0
MOVL C01179 V=800.0 PL=0
MOVL C01180 V=800.0 PL=0
MOVL C01181 V=800.0 PL=0
MOVL C01182 V=800.0 PL=0
MOVL C01183 V=800.0 PL=0
MOVL C01184 V=800.0 PL=0
MOVL C01185 V=800.0 PL=0
MOVL C01186 V=800.0 PL=0
MOVL C01187 V=800.0 PL=0
MOVL C01188 V=800.0 PL=0
MOVL C01189 V=800.0 PL=0
MOVL C01190 V=800.0 PL=0
MOVL C01191 V=800.0 PL=0
MOVL C01192 V=800.0 PL=0
MOVL C01193 V=800.0 PL=0
MOVL C01194 V=800.0 PL=0
MOVL C01195 V=800.0 PL=0
MOVL C01196 V=800.0 PL=0
MOVL C01197 V=800.0 PL=0
MOVL C01198 V=800.0 PL=0
MOVL C01199 V=800.0 PL=0
MOVL C01200 V=800.0 PL=0
MOVL C01201 V=800.0 PL=0
MOVL C01202 V=800.0 PL=0
MOVL C01203 V=800.0 PL=0
MOVL C01204 V=800.0 PL=0
MOVL C01205 V=800.0 PL=0
MOVL C01206 V=800.0 PL=0
MOVL C01207 V=800.0 PL=0
MOVL C01208 V=800.0 PL=0
MOVL C01209 V=800.0 PL=0
MOVL C01210 V=800.0 PL=0
MOVL C01211 V=800.0 PL=0
MOVL C01212 V=800.0 PL=0
MOVL C01213 V=800.0 PL=0
MOVL C01214 V=800.0 PL=0
MOVL C01215 V=800.0 PL=0
MOVL C01216 V=800.0 PL=0
MOVL C01217 V=800.0 PL=0
MOVL C01218 V=800.0 PL=0
MOVL C01219 V=800.0 PL=0
MOVL C01220 V=800.0 PL=0
MOVL C01221 V=800.0 PL=0
MOVL C01222 V=800.0 PL=0
MOVL C01223 V=800.0 PL=0
MOVL C01224 V=800.0 PL=0
MOVL C01225 V=800.0 PL=0
MOVL C01226 V=800.0 PL=0
MOVL C01227 V=800.0 PL=0
MOVL C01228 V=800.0 PL=0
MOVL C01229 V=800.0 PL=0
MOVL C01230 V=800.0 PL=0
MOVL C01231 V=800.0 PL=0
MOVL C01232 V=800.0 PL=0
MOVL C01233 V=800.0 PL=0
MOVL C01234 V=800.0 PL=0
MOVL C01235 V=800.0 PL=0
MOVL C01236 V=800.0 PL=0
MOVL C01237 V=800.0 PL=0
MOVL C01238 V=800.0 PL=0
MOVL C01239 V=800.0 PL=0
MOVL C01240 V=800.0 PL=0
MOVL C01241 V=800.0 PL=0
MOVL C01242 V=800.0 PL=0
MOVL C01243 V=800.0 PL=0
MOVL C01244 V=800.0 PL=0
MOVL C01245 V=800.0 PL=0
MOVL C01246 V=800.0 PL=0
MOVL C01247 V=800.0 PL=0
MOVL C01248 V=800.0 PL=0
MOVL C01249 V=800.0 PL=0
MOVL C01250 V=800.0 PL=0
MOVL C01251 V=800.0 PL=0
MOVL C01252 V=800.0 PL=0
MOVL C01253 V=800.0 PL=0
MOVL C01254 V=800.0 PL=0
MOVL C01255 V=800.0 PL=0
MOVL C01256 V=800.0 PL=0
MOVL C01257 V=800.0 PL=0
MOVL C01258 V=800.0 PL=0
MOVL C01259 V=800.0 PL=0
MOVL C01260 V=800.0 PL=0
MOVL C01261 V=800.0 PL=0
MOVL C01262 V=800.0 PL=0
MOVL C01263 V=800.0 PL=0
MOVL C01264 V=800.0 PL=0
MOVL C01265 V=800.0 PL=0
MOVL C01266 V=800.0 PL=0
MOVL C01267 V=800.0 PL=0
MOVL C01268 V=800.0 PL=0
MOVL C01269 V=800.0 PL=0
MOVL C01270 V=800.0 PL=0
MOVL C01271 V=800.0 PL=0
MOVL C01272 V=800.0 PL=0
MOVL C01273 V=800.0 PL=0
MOVL C01274 V=800.0 PL=0
MOVL C01275 V=800.0 PL=0
MOVL C01276 V=800.0 PL=0
MOVL C01277 V=800.0 PL=0
MOVL C01278 V=800.0 PL=0
MOVL C01279 V=800.0 PL=0
MOVL C01280 V=800.0 PL=0
MOVL C01281 V=800.0 PL=0
MOVL C01282 V=800.0 PL=0
MOVL C01283 V=800.0 PL=0
MOVL C01284 V=800.0 PL=0
MOVL C01285 V=800.0 PL=0
MOVL C01286 V=800.0 PL=0
MOVL C01287 V=800.0 PL=0
MOVL C01288 V=800.0 PL=0
MOVL C01289 V=800.0 PL=0
MOVL C01290 V=800.0 PL=0
MOVL C01291 V=800.0 PL=0
MOVL C01292 V=800.0 PL=0
MOVL C01293 V=800.0 PL=0
MOVL C01294 V=800.0 PL=0
MOVL C01295 V=800.0 PL=0
MOVL C01296 V=800.0 PL=0
MOVL C01297 V=800.0 PL=0
MOVL C01298 V=800.0 PL=0
MOVL C01299 V=800.0 PL=0
MOVL C01300 V=800.0 PL=0
MOVL C01301 V=800.0 PL=0
MOVL C01302 V=800.0 PL=0
MOVL C01303 V=800.0 PL=0
MOVL C01304 V=800.0 PL=0
MOVL C01305 V=800.0 PL=0
MOVL C01306 V=800.0 PL=0
MOVL C01307 V=800.0 PL=0
MOVL C01308 V=800.0 PL=0
MOVL C01309 V=800.0 PL=0
MOVL C01310 V=800.0 PL=0
MOVL C01311 V=800.0 PL=0
MOVL C01312 V=800.0 PL=0
MOVL C01313 V=800.0 PL=0
MOVL C01314 V=800.0 PL=0
MOVL C01315 V=800.0 PL=0
MOVL C01316 V=800.0 PL=0
MOVL C01317 V=800.0 PL=0
MOVL C01318 V=800.0 PL=0
MOVL C01319 V=800.0 PL=0
MOVL C01320 V=800.0 PL=0
MOVL C01321 V=800.0 PL=0
MOVL C01322 V=800.0 PL=0
MOVL C01323 V=800.0 PL=0
MOVL C01324 V=800.0 PL=0
MOVL C01325 V=800.0 PL=0
MOVL C01326 V=800.0 PL=0
MOVL C01327 V=800.0 PL=0
MOVL C01328 V=800.0 PL=0
MOVL C01329 V=800.0 PL=0
MOVL C01330 V=800.0 PL=0
MOVL C01331 V=800.0 PL=0
MOVL C01332 V=800.0 PL=0
MOVL C01333 V=800.0 PL=0
MOVL C01334 V=800.0 PL=0
MOVL C01335 V=800.0 PL=0
MOVL C01336 V=800.0 PL=0
MOVL C01337 V=800.0 PL=0
MOVL C01338 V=800.0 PL=0
MOVL C01339 V=800.0 PL=0
MOVL C01340 V=800.0 PL=0
MOVL C01341 V=800.0 PL=0
MOVL C01342 V=800.0 PL=0
MOVL C01343 V=800.0 PL=0
MOVL C01344 V=800.0 PL=0
MOVL C01345 V=800.0 PL=0
MOVL C01346 V=800.0 PL=0
MOVL C01347 V=800.0 PL=0
MOVL C01348 V=800.0 PL=0
MOVL C01349 V=800.0 PL=0
MOVL C01350 V=800.0 PL=0
MOVL C01351 V=800.0 PL=0
MOVL C01352 V=800.0 PL=0
MOVL C01353 V=800.0 PL=0
MOVL C01354 V=800.0 PL=0
MOVL C01355 V=800.0 PL=0
MOVL C01356 V=800.0 PL=0
MOVL C01357 V=800.0 PL=0
MOVL C01358 V=800.0 PL=0
MOVL C01359 V=800.0 PL=0
MOVL C01360 V=800.0 PL=0
MOVL C01361 V=800.0 PL=0
MOVL C01362 V=800.0 PL=0
MOVL C01363 V=800.0 PL=0
MOVL C01364 V=800.0 PL=0
MOVL C01365 V=800.0 PL=0
MOVL C01366 V=800.0 PL=0
MOVL C01367 V=800.0 PL=0
MOVL C01368 V=800.0 PL=0
MOVL C01369 V=800.0 PL=0
MOVL C01370 V=800.0 PL=0
MOVL C01371 V=800.0 PL=0
MOVL C01372 V=800.0 PL=0
MOVL C01373 V=800.0 PL=0
MOVL C01374 V=800.0 PL=0
MOVL C01375 V=800.0 PL=0
MOVL C01376 V=800.0 PL=0
MOVL C01377 V=800.0 PL=0
MOVL C01378 V=800.0 PL=0
MOVL C01379 V=800.0 PL=0
MOVL C01380 V=800.0 PL=0
MOVL C01381 V=800.0 PL=0
MOVL C01382 V=800.0 PL=0
MOVL C01383 V=800.0 PL=0
MOVL C01384 V=800.0 PL=0
MOVL C01385 V=800.0 PL=0
MOVL C01386 V=800.0 PL=0
MOVL C01387 V=800.0 PL=0
MOVL C01388 V=800.0 PL=0
MOVL C01389 V=800.0 PL=0
MOVL C01390 V=800.0 PL=0
MOVL C01391 V=800.0 PL=0
MOVL C01392 V=800.0 PL=0
MOVL C01393 V=800.0 PL=0
MOVL C01394 V=800.0 PL=0
MOVL C01395 V=800.0 PL=0
MOVL C01396 V=800.0 PL=0
MOVL C01397 V=800.0 PL=0
MOVL C01398 V=800.0 PL=0
MOVL C01399 V=800.0 PL=0
MOVL C01400 V=800.0 PL=0
MOVL C01401 V=800.0 PL=0
MOVL C01402 V=800.0 PL=0
MOVL C01403 V=800.0 PL=0
MOVL C01404 V=800.0 PL=0
MOVL C01405 V=800.0 PL=0
MOVL C01406 V=800.0 PL=0
MOVL C01407 V=800.0 PL=0
MOVL C01408 V=800.0 PL=0
MOVL C01409 V=800.0 PL=0
MOVL C01410 V=800.0 PL=0
MOVL C01411 V=800.0 PL=0
MOVL C01412 V=800.0 PL=0
MOVL C01413 V=800.0 PL=0
MOVL C01414 V=800.0 PL=0
MOVL C01415 V=800.0 PL=0
MOVL C01416 V=800.0 PL=0
MOVL C01417 V=800.0 PL=0
MOVL C01418 V=800.0 PL=0
MOVL C01419 V=800.0 PL=0
MOVL C01420 V=800.0 PL=0
MOVL C01421 V=800.0 PL=0
MOVL C01422 V=800.0 PL=0
MOVL C01423 V=800.0 PL=0
MOVL C01424 V=800.0 PL=0
MOVL C01425 V=800.0 PL=0
MOVL C01426 V=800.0 PL=0
MOVL C01427 V=800.0 PL=0
MOVL C01428 V=800.0 PL=0
MOVL C01429 V=800.0 PL=0
MOVL C01430 V=800.0 PL=0
MOVL C01431 V=800.0 PL=0
MOVL C01432 V=800.0 PL=0
MOVL C01433 V=800.0 PL=0
MOVL C01434 V=800.0 PL=0
MOVL C01435 V=800.0 PL=0
MOVL C01436 V=800.0 PL=0
MOVL C01437 V=800.0 PL=0
MOVL C01438 V=800.0 PL=0
MOVL C01439 V=800.0 PL=0
MOVL C01440 V=800.0 PL=0
MOVL C01441 V=800.0 PL=0
MOVL C01442 V=800.0 PL=0
MOVL C01443 V=800.0 PL=0
MOVL C01444 V=800.0 PL=0
MOVL C01445 V=800.0 PL=0
MOVL C01446 V=800.0 PL=0
MOVL C01447 V=800.0 PL=0
MOVL C01448 V=800.0 PL=0
MOVL C01449 V=800.0 PL=0
MOVL C01450 V=800.0 PL=0
MOVL C01451 V=800.0 PL=0
MOVL C01452 V=800.0 PL=0
MOVL C01453 V=800.0 PL=0
MOVL C01454 V=800.0 PL=0
MOVL C01455 V=800.0 PL=0
MOVL C01456 V=800.0 PL=0
MOVL C01457 V=800.0 PL=0
MOVL C01458 V=800.0 PL=0
MOVL C01459 V=800.0 PL=0
MOVL C01460 V=800.0 PL=0
MOVL C01461 V=800.0 PL=0
MOVL C01462 V=800.0 PL=0
MOVL C01463 V=800.0 PL=0
MOVL C01464 V=800.0 PL=0
MOVL C01465 V=800.0 PL=0
MOVL C01466 V=800.0 PL=0
MOVL C01467 V=800.0 PL=0
MOVL C01468 V=800.0 PL=0
MOVL C01469 V=800.0 PL=0
MOVL C01470 V=800.0 PL=0
MOVL C01471 V=800.0 PL=0
MOVL C01472 V=800.0 PL=0
MOVL C01473 V=800.0 PL=0
MOVL C01474 V=800.0 PL=0
MOVL C01475 V=800.0 PL=0
MOVL C01476 V=800.0 PL=0
MOVL C01477 V=800.0 PL=0
MOVL C01478 V=800.0 PL=0
MOVL C01479 V=800.0 PL=0
MOVL C01480 V=800.0 PL=0
MOVL C01481 V=800.0 PL=0
MOVL C01482 V=800.0 PL=0
MOVL C01483 V=800.0 PL=0
MOVL C01484 V=800.0 PL=0
MOVL C01485 V=800.0 PL=0
MOVL C01486 V=800.0 PL=0
MOVL C01487 V=800.0 PL=0
MOVL C01488 V=800.0 PL=0
MOVL C01489 V=800.0 PL=0
MOVL C01490 V=800.0 PL=0
MOVL C01491 V=800.0 PL=0
MOVL C01492 V=800.0 PL=0
MOVL C01493 V=800.0 PL=0
MOVL C01494 V=800.0 PL=0
MOVL C01495 V=800.0 PL=0
MOVL C01496 V=800.0 PL=0
MOVL C01497 V=800.0 PL=0
MOVL C01498 V=800.0 PL=0
MOVL C01499 V=800.0 PL=0
MOVL C01500 V=800.0 PL=0
MOVL C01501 V=800.0 PL=0
MOVL C01502 V=800.0 PL=0
MOVL C01503 V=800.0 PL=0
MOVL C01504 V=800.0 PL=0
MOVL C01505 V=800.0 PL=0
MOVL C01506 V=800.0 PL=0
MOVL C01507 V=800.0 PL=0
MOVL C01508 V=800.0 PL=0
MOVL C01509 V=800.0 PL=0
MOVL C01510 V=800.0 PL=0
MOVL C01511 V=800.0 PL=0
MOVL C01512 V=800.0 PL=0
MOVL C01513 V=800.0 PL=0
MOVL C01514 V=800.0 PL=0
MOVL C01515 V=800.0 PL=0
MOVL C01516 V=800.0 PL=0
MOVL C01517 V=800.0 PL=0
MOVL C01518 V=800.0 PL=0
MOVL C01519 V=800.0 PL=0
MOVL C01520 V=800.0 PL=0
MOVL C01521 V=800.0 PL=0
MOVL C01522 V=800.0 PL=0
MOVL C01523 V=800.0 PL=0
MOVL C01524 V=800.0 PL=0
MOVL C01525 V=800.0 PL=0
MOVL C01526 V=800.0 PL=0
MOVL C01527 V=800.0 PL=0
MOVL C01528 V=800.0 PL=0
MOVL C01529 V=800.0 PL=0
MOVL C01530 V=800.0 PL=0
MOVL C01531 V=800.0 PL=0
MOVL C01532 V=800.0 PL=0
MOVL C01533 V=800.0 PL=0
MOVL C01534 V=800.0 PL=0
MOVL C01535 V=800.0 PL=0
MOVL C01536 V=800.0 PL=0
MOVL C01537 V=800.0 PL=0
MOVL C01538 V=800.0 PL=0
MOVL C01539 V=800.0 PL=0
MOVL C01540 V=800.0 PL=0
MOVL C01541 V=800.0 PL=0
MOVL C01542 V=800.0 PL=0
MOVL C01543 V=800.0 PL=0
MOVL C01544 V=800.0 PL=0
MOVL C01545 V=800.0 PL=0
MOVL C01546 V=800.0 PL=0
MOVL C01547 V=800.0 PL=0
MOVL C01548 V=800.0 PL=0
MOVL C01549 V=800.0 PL=0
MOVL C01550 V=800.0 PL=0
MOVL C01551 V=800.0 PL=0
MOVL C01552 V=800.0 PL=0
MOVL C01553 V=800.0 PL=0
MOVL C01554 V=800.0 PL=0
MOVL C01555 V=800.0 PL=0
MOVL C01556 V=800.0 PL=0
MOVL C01557 V=800.0 PL=0
MOVL C01558 V=800.0 PL=0
MOVL C01559 V=800.0 PL=0
MOVL C01560 V=800.0 PL=0
MOVL C01561 V=800.0 PL=0
MOVL C01562 V=800.0 PL=0
MOVL C01563 V=800.0 PL=0
MOVL C01564 V=800.0 PL=0
MOVL C01565 V=800.0 PL=0
MOVL C01566 V=800.0 PL=0
MOVL C01567 V=800.0 PL=0
MOVL C01568 V=800.0 PL=0
MOVL C01569 V=800.0 PL=0
MOVL C01570 V=800.0 PL=0
MOVL C01571 V=800.0 PL=0
MOVL C01572 V=800.0 PL=0
MOVL C01573 V=800.0 PL=0
MOVL C01574 V=800.0 PL=0
MOVL C01575 V=800.0 PL=0
MOVL C01576 V=800.0 PL=0
MOVL C01577 V=800.0 PL=0
MOVL C01578 V=800.0 PL=0
MOVL C01579 V=800.0 PL=0
MOVL C01580 V=800.0 PL=0
MOVL C01581 V=800.0 PL=0
MOVL C01582 V=800.0 PL=0
MOVL C01583 V=800.0 PL=0
MOVL C01584 V=800.0 PL=0
MOVL C01585 V=800.0 PL=0
MOVL C01586 V=800.0 PL=0
MOVL C01587 V=800.0 PL=0
MOVL C01588 V=800.0 PL=0
MOVL C01589 V=800.0 PL=0
MOVL C01590 V=800.0 PL=0
MOVL C01591 V=800.0 PL=0
MOVL C01592 V=800.0 PL=0
MOVL C01593 V=800.0 PL=0
MOVL C01594 V=800.0 PL=0
MOVL C01595 V=800.0 PL=0
MOVL C01596 V=800.0 PL=0
MOVL C01597 V=800.0 PL=0
MOVL C01598 V=800.0 PL=0
MOVL C01599 V=800.0 PL=0
MOVL C01600 V=800.0 PL=0
MOVL C01601 V=800.0 PL=0
MOVL C01602 V=800.0 PL=0
MOVL C01603 V=800.0 PL=0
MOVL C01604 V=800.0 PL=0
MOVL C01605 V=800.0 PL=0
MOVL C01606 V=800.0 PL=0
MOVL C01607 V=800.0 PL=0
MOVL C01608 V=800.0 PL=0
MOVL C01609 V=800.0 PL=0
MOVL C01610 V=800.0 PL=0
MOVL C01611 V=800.0 PL=0
MOVL C01612 V=800.0 PL=0
MOVL C01613 V=800.0 PL=0
MOVL C01614 V=800.0 PL=0
MOVL C01615 V=800.0 PL=0
MOVL C01616 V=800.0 PL=0
MOVL C01617 V=800.0 PL=0
MOVL C01618 V=800.0 PL=0
MOVL C01619 V=800.0 PL=0
MOVL C01620 V=800.0 PL=0
MOVL C01621 V=800.0 PL=0
MOVL C01622 V=800.0 PL=0
MOVL C01623 V=800.0 PL=0
MOVL C01624 V=800.0 PL=0
MOVL C01625 V=800.0 PL=0
MOVL C01626 V=800.0 PL=0
MOVL C01627 V=800.0 PL=0
MOVL C01628 V=800.0 PL=0
MOVL C01629 V=800.0 PL=0
MOVL C01630 V=800.0 PL=0
MOVL C01631 V=800.0 PL=0
MOVL C01632 V=800.0 PL=0
MOVL C01633 V=800.0 PL=0
MOVL C01634 V=800.0 PL=0
MOVL C01635 V=800.0 PL=0
MOVL C01636 V=800.0 PL=0
MOVL C01637 V=800.0 PL=0
MOVL C01638 V=800.0 PL=0
MOVL C01639 V=800.0 PL=0
MOVL C01640 V=800.0 PL=0
MOVL C01641 V=800.0 PL=0
MOVL C01642 V=800.0 PL=0
MOVL C01643 V=800.0 PL=0
MOVL C01644 V=800.0 PL=0
MOVL C01645 V=800.0 PL=0
MOVL C01646 V=800.0 PL=0
MOVL C01647 V=800.0 PL=0
MOVL C01648 V=800.0 PL=0
MOVL C01649 V=800.0 PL=0
MOVL C01650 V=800.0 PL=0
MOVL C01651 V=800.0 PL=0
MOVL C01652 V=800.0 PL=0
MOVL C01653 V=800.0 PL=0
MOVL C01654 V=800.0 PL=0
MOVL C01655 V=800.0 PL=0
MOVL C01656 V=800.0 PL=0
MOVL C01657 V=800.0 PL=0
MOVL C01658 V=800.0 PL=0
MOVL C01659 V=800.0 PL=0
MOVL C01660 V=800.0 PL=0
MOVL C01661 V=800.0 PL=0
MOVL C01662 V=800.0 PL=0
MOVL C01663 V=800.0 PL=0
MOVL C01664 V=800.0 PL=0
MOVL C01665 V=800.0 PL=0
MOVL C01666 V=800.0 PL=0
MOVL C01667 V=800.0 PL=0
MOVL C01668 V=800.0 PL=0
MOVL C01669 V=800.0 PL=0
MOVL C01670 V=800.0 PL=0
MOVL C01671 V=800.0 PL=0
MOVL C01672 V=800.0 PL=0
MOVL C01673 V=800.0 PL=0
MOVL C01674 V=800.0 PL=0
MOVL C01675 V=800.0 PL=0
MOVL C01676 V=800.0 PL=0
MOVL C01677 V=800.0 PL=0
MOVL C01678 V=800.0 PL=0
MOVL C01679 V=800.0 PL=0
MOVL C01680 V=800.0 PL=0
MOVL C01681 V=800.0 PL=0
MOVL C01682 V=800.0 PL=0
MOVL C01683 V=800.0 PL=0
MOVL C01684 V=800.0 PL=0
MOVL C01685 V=800.0 PL=0
MOVL C01686 V=800.0 PL=0
MOVL C01687 V=800.0 PL=0
MOVL C01688 V=800.0 PL=0
MOVL C01689 V=800.0 PL=0
MOVL C01690 V=800.0 PL=0
MOVL C01691 V=800.0 PL=0
MOVL C01692 V=800.0 PL=0
MOVL C01693 V=800.0 PL=0
MOVL C01694 V=800.0 PL=0
MOVL C01695 V=800.0 PL=0
MOVL C01696 V=800.0 PL=0
MOVL C01697 V=800.0 PL=0
MOVL C01698 V=800.0 PL=0
MOVL C01699 V=800.0 PL=0
MOVL C01700 V=800.0 PL=0
MOVL C01701 V=800.0 PL=0
MOVL C01702 V=800.0 PL=0
MOVL C01703 V=800.0 PL=0
MOVL C01704 V=800.0 PL=0
MOVL C01705 V=800.0 PL=0
MOVL C01706 V=800.0 PL=0
MOVL C01707 V=800.0 PL=0
MOVL C01708 V=800.0 PL=0
MOVL C01709 V=800.0 PL=0
MOVL C01710 V=800.0 PL=0
MOVL C01711 V=800.0 PL=0
MOVL C01712 V=800.0 PL=0
MOVL C01713 V=800.0 PL=0
MOVL C01714 V=800.0 PL=0
MOVL C01715 V=800.0 PL=0
MOVL C01716 V=800.0 PL=0
MOVL C01717 V=800.0 PL=0
MOVL C01718 V=800.0 PL=0
MOVL C01719 V=800.0 PL=0
MOVL C01720 V=800.0 PL=0
MOVL C01721 V=800.0 PL=0
MOVL C01722 V=800.0 PL=0
MOVL C01723 V=800.0 PL=0
MOVL C01724 V=800.0 PL=0
MOVL C01725 V=800.0 PL=0
MOVL C01726 V=800.0 PL=0
MOVL C01727 V=800.0 PL=0
MOVL C01728 V=800.0 PL=0
MOVL C01729 V=800.0 PL=0
MOVL C01730 V=800.0 PL=0
MOVL C01731 V=800.0 PL=0
MOVL C01732 V=800.0 PL=0
MOVL C01733 V=800.0 PL=0
MOVL C01734 V=800.0 PL=0
MOVL C01735 V=800.0 PL=0
MOVL C01736 V=800.0 PL=0
MOVL C01737 V=800.0 PL=0
MOVL C01738 V=800.0 PL=0
MOVL C01739 V=800.0 PL=0
MOVL C01740 V=800.0 PL=0
MOVL C01741 V=800.0 PL=0
MOVL C01742 V=800.0 PL=0
MOVL C01743 V=800.0 PL=0
MOVL C01744 V=800.0 PL=0
MOVL C01745 V=800.0 PL=0
MOVL C01746 V=800.0 PL=0
MOVL C01747 V=800.0 PL=0
MOVL C01748 V=800.0 PL=0
MOVL C01749 V=800.0 PL=0
MOVL C01750 V=800.0 PL=0
MOVL C01751 V=800.0 PL=0
MOVL C01752 V=800.0 PL=0
MOVL C01753 V=800.0 PL=0
MOVL C01754 V=800.0 PL=0
MOVL C01755 V=800.0 PL=0
MOVL C01756 V=800.0 PL=0
MOVL C01757 V=800.0 PL=0
MOVL C01758 V=800.0 PL=0
MOVL C01759 V=800.0 PL=0
MOVL C01760 V=800.0 PL=0
MOVL C01761 V=800.0 PL=0
MOVL C01762 V=800.0 PL=0
MOVL C01763 V=800.0 PL=0
MOVL C01764 V=800.0 PL=0
MOVL C01765 V=800.0 PL=0
MOVL C01766 V=800.0 PL=0
MOVL C01767 V=800.0 PL=0
MOVL C01768 V=800.0 PL=0
MOVL C01769 V=800.0 PL=0
MOVL C01770 V=800.0 PL=0
MOVL C01771 V=800.0 PL=0
MOVL C01772 V=800.0 PL=0
MOVL C01773 V=800.0 PL=0
MOVL C01774 V=800.0 PL=0
MOVL C01775 V=800.0 PL=0
MOVL C01776 V=800.0 PL=0
MOVL C01777 V=800.0 PL=0
MOVL C01778 V=800.0 PL=0
MOVL C01779 V=800.0 PL=0
MOVL C01780 V=800.0 PL=0
MOVL C01781 V=800.0 PL=0
MOVL C01782 V=800.0 PL=0
MOVL C01783 V=800.0 PL=0
MOVL C01784 V=800.0 PL=0
MOVL C01785 V=800.0 PL=0
MOVL C01786 V=800.0 PL=0
MOVL C01787 V=800.0 PL=0
MOVL C01788 V=800.0 PL=0
MOVL C01789 V=800.0 PL=0
MOVL C01790 V=800.0 PL=0
MOVL C01791 V=800.0 PL=0
MOVL C01792 V=800.0 PL=0
MOVL C01793 V=800.0 PL=0
MOVL C01794 V=800.0 PL=0
MOVL C01795 V=800.0 PL=0
MOVL C01796 V=800.0 PL=0
MOVL C01797 V=800.0 PL=0
MOVL C01798 V=800.0 PL=0
MOVL C01799 V=800.0 PL=0
MOVL C01800 V=800.0 PL=0
MOVL C01801 V=800.0 PL=0
MOVL C01802 V=800.0 PL=0
MOVL C01803 V=800.0 PL=0
MOVL C01804 V=800.0 PL=0
MOVL C01805 V=800.0 PL=0
MOVL C01806 V=800.0 PL=0
MOVL C01807 V=800.0 PL=0
MOVL C01808 V=800.0 PL=0
MOVL C01809 V=800.0 PL=0
MOVL C01810 V=800.0 PL=0
MOVL C01811 V=800.0 PL=0
MOVL C01812 V=800.0 PL=0
MOVL C01813 V=800.0 PL=0
MOVL C01814 V=800.0 PL=0
MOVL C01815 V=800.0 PL=0
MOVL C01816 V=800.0 PL=0
MOVL C01817 V=800.0 PL=0
MOVL C01818 V=800.0 PL=0
MOVL C01819 V=800.0 PL=0
MOVL C01820 V=800.0 PL=0
MOVL C01821 V=800.0 PL=0
MOVL C01822 V=800.0 PL=0
MOVL C01823 V=800.0 PL=0
MOVL C01824 V=800.0 PL=0
MOVL C01825 V=800.0 PL=0
MOVL C01826 V=800.0 PL=0
MOVL C01827 V=800.0 PL=0
MOVL C01828 V=800.0 PL=0
MOVL C01829 V=800.0 PL=0
MOVL C01830 V=800.0 PL=0
MOVL C01831 V=800.0 PL=0
MOVL C01832 V=800.0 PL=0
MOVL C01833 V=800.0 PL=0
MOVL C01834 V=800.0 PL=0
MOVL C01835 V=800.0 PL=0
MOVL C01836 V=800.0 PL=0
MOVL C01837 V=800.0 PL=0
MOVL C01838 V=800.0 PL=0
MOVL C01839 V=800.0 PL=0
MOVL C01840 V=800.0 PL=0
MOVL C01841 V=800.0 PL=0
MOVL C01842 V=800.0 PL=0
MOVL C01843 V=800.0 PL=0
MOVL C01844 V=800.0 PL=0
MOVL C01845 V=800.0 PL=0
MOVL C01846 V=800.0 PL=0
MOVL C01847 V=800.0 PL=0
MOVL C01848 V=800.0 PL=0
MOVL C01849 V=800.0 PL=0
MOVL C01850 V=800.0 PL=0
MOVL C01851 V=800.0 PL=0
MOVL C01852 V=800.0 PL=0
MOVL C01853 V=800.0 PL=0
MOVL C01854 V=800.0 PL=0
MOVL C01855 V=800.0 PL=0
MOVL C01856 V=800.0 PL=0
MOVL C01857 V=800.0 PL=0
MOVL C01858 V=800.0 PL=0
MOVL C01859 V=800.0 PL=0
MOVL C01860 V=800.0 PL=0
MOVL C01861 V=800.0 PL=0
MOVL C01862 V=800.0 PL=0
MOVL C01863 V=800.0 PL=0
MOVL C01864 V=800.0 PL=0
MOVL C01865 V=800.0 PL=0
MOVL C01866 V=800.0 PL=0
MOVL C01867 V=800.0 PL=0
MOVL C01868 V=800.0 PL=0
MOVL C01869 V=800.0 PL=0
MOVL C01870 V=800.0 PL=0
MOVL C01871 V=800.0 PL=0
MOVL C01872 V=800.0 PL=0
MOVL C01873 V=800.0 PL=0
MOVL C01874 V=800.0 PL=0
MOVL C01875 V=800.0 PL=0
MOVL C01876 V=800.0 PL=0
MOVL C01877 V=800.0 PL=0
MOVL C01878 V=800.0 PL=0
MOVL C01879 V=800.0 PL=0
MOVL C01880 V=800.0 PL=0
MOVL C01881 V=800.0 PL=0
MOVL C01882 V=800.0 PL=0
MOVL C01883 V=800.0 PL=0
MOVL C01884 V=800.0 PL=0
MOVL C01885 V=800.0 PL=0
MOVL C01886 V=800.0 PL=0
MOVL C01887 V=800.0 PL=0
MOVL C01888 V=800.0 PL=0
MOVL C01889 V=800.0 PL=0
MOVL C01890 V=800.0 PL=0
MOVL C01891 V=800.0 PL=0
MOVL C01892 V=800.0 PL=0
MOVL C01893 V=800.0 PL=0
MOVL C01894 V=800.0 PL=0
MOVL C01895 V=800.0 PL=0
MOVL C01896 V=800.0 PL=0
MOVL C01897 V=800.0 PL=0
MOVL C01898 V=800.0 PL=0
MOVL C01899 V=800.0 PL=0
MOVL C01900 V=800.0 PL=0
MOVL C01901 V=800.0 PL=0
MOVL C01902 V=800.0 PL=0
MOVL C01903 V=800.0 PL=0
MOVL C01904 V=800.0 PL=0
MOVL C01905 V=800.0 PL=0
MOVL C01906 V=800.0 PL=0
MOVL C01907 V=800.0 PL=0
MOVL C01908 V=800.0 PL=0
MOVL C01909 V=800.0 PL=0
MOVL C01910 V=800.0 PL=0
MOVL C01911 V=800.0 PL=0
MOVL C01912 V=800.0 PL=0
MOVL C01913 V=800.0 PL=0
MOVL C01914 V=800.0 PL=0
MOVL C01915 V=800.0 PL=0
MOVL C01916 V=800.0 PL=0
MOVL C01917 V=800.0 PL=0
MOVL C01918 V=800.0 PL=0
MOVL C01919 V=800.0 PL=0
MOVL C01920 V=800.0 PL=0
MOVL C01921 V=800.0 PL=0
MOVL C01922 V=800.0 PL=0
MOVL C01923 V=800.0 PL=0
MOVL C01924 V=800.0 PL=0
MOVL C01925 V=800.0 PL=0
MOVL C01926 V=800.0 PL=0
MOVL C01927 V=800.0 PL=0
MOVL C01928 V=800.0 PL=0
MOVL C01929 V=800.0 PL=0
MOVL C01930 V=800.0 PL=0
MOVL C01931 V=800.0 PL=0
MOVL C01932 V=800.0 PL=0
MOVL C01933 V=800.0 PL=0
MOVL C01934 V=800.0 PL=0
MOVL C01935 V=800.0 PL=0
MOVL C01936 V=800.0 PL=0
MOVL C01937 V=800.0 PL=0
MOVL C01938 V=800.0 PL=0
MOVL C01939 V=800.0 PL=0
MOVL C01940 V=800.0 PL=0
MOVL C01941 V=800.0 PL=0
MOVL C01942 V=800.0 PL=0
MOVL C01943 V=800.0 PL=0
MOVL C01944 V=800.0 PL=0
MOVL C01945 V=800.0 PL=0
MOVL C01946 V=800.0 PL=0
MOVL C01947 V=800.0 PL=0
MOVL C01948 V=800.0 PL=0
MOVL C01949 V=800.0 PL=0
MOVL C01950 V=800.0 PL=0
MOVL C01951 V=800.0 PL=0
MOVL C01952 V=800.0 PL=0
MOVL C01953 V=800.0 PL=0
MOVL C01954 V=800.0 PL=0
MOVL C01955 V=800.0 PL=0
MOVL C01956 V=800.0 PL=0
MOVL C01957 V=800.0 PL=0
MOVL C01958 V=800.0 PL=0
MOVL C01959 V=800.0 PL=0
MOVL C01960 V=800.0 PL=0
MOVL C01961 V=800.0 PL=0
MOVL C01962 V=800.0 PL=0
MOVL C01963 V=800.0 PL=0
MOVL C01964 V=800.0 PL=0
MOVL C01965 V=800.0 PL=0
MOVL C01966 V=800.0 PL=0
MOVL C01967 V=800.0 PL=0
MOVL C01968 V=800.0 PL=0
MOVL C01969 V=800.0 PL=0
MOVL C01970 V=800.0 PL=0
MOVL C01971 V=800.0 PL=0
MOVL C01972 V=800.0 PL=0
MOVL C01973 V=800.0 PL=0
MOVL C01974 V=800.0 PL=0
MOVL C01975 V=800.0 PL=0
MOVL C01976 V=800.0 PL=0
MOVL C01977 V=800.0 PL=0
MOVL C01978 V=800.0 PL=0
MOVL C01979 V=800.0 PL=0
MOVL C01980 V=800.0 PL=0
MOVL C01981 V=800.0 PL=0
MOVL C01982 V=800.0 PL=0
MOVL C01983 V=800.0 PL=0
MOVL C01984 V=800.0 PL=0
MOVL C01985 V=800.0 PL=0
MOVL C01986 V=800.0 PL=0
MOVL C01987 V=800.0 PL=0
MOVL C01988 V=800.0 PL=0
MOVL C01989 V=800.0 PL=0
MOVL C01990 V=800.0 PL=0
MOVL C01991 V=800.0 PL=0
MOVL C01992 V=800.0 PL=0
MOVL C01993 V=800.0 PL=0
MOVL C01994 V=800.0 PL=0
MOVL C01995 V=800.0 PL=0
MOVL C01996 V=800.0 PL=0
MOVL C01997 V=800.0 PL=0
MOVL C01998 V=800.0 PL=0
MOVL C01999 V=800.0 PL=0
MOVL C02000 V=800.0 PL=0
MOVL C02001 V=800.0 PL=0
MOVL C02002 V=800.0 PL=0
MOVL C02003 V=800.0 PL=0
MOVL C02004 V=800.0 PL=0
MOVL C02005 V=800.0 PL=0
MOVL C02006 V=800.0 PL=0
MOVL C02007 V=800.0 PL=0
MOVL C02008 V=800.0 PL=0
MOVL C02009 V=800.0 PL=0
MOVL C02010 V=800.0 PL=0
MOVL C02011 V=800.0 PL=0
MOVL C02012 V=800.0 PL=0
MOVL C02013 V=800.0 PL=0
MOVL C02014 V=800.0 PL=0
MOVL C02015 V=800.0 PL=0
MOVL C02016 V=800.0 PL=0
MOVL C02017 V=800.0 PL=0
MOVL C02018 V=800.0 PL=0
MOVL C02019 V=800.0 PL=0
MOVL C02020 V=800.0 PL=0
MOVL C02021 V=800.0 PL=0
MOVL C02022 V=800.0 PL=0
MOVL C02023 V=800.0 PL=0
MOVL C02024 V=800.0 PL=0
MOVL C02025 V=800.0 PL=0
MOVL C02026 V=800.0 PL=0
MOVL C02027 V=800.0 PL=0
MOVL C02028 V=800.0 PL=0
MOVL C02029 V=800.0 PL=0
MOVL C02030 V=800.0 PL=0
MOVL C02031 V=800.0 PL=0
MOVL C02032 V=800.0 PL=0
MOVL C02033 V=800.0 PL=0
MOVL C02034 V=800.0 PL=0
MOVL C02035 V=800.0 PL=0
MOVL C02036 V=800.0 PL=0
MOVL C02037 V=800.0 PL=0
MOVL C02038 V=800.0 PL=0
MOVL C02039 V=800.0 PL=0
MOVL C02040 V=800.0 PL=0
MOVL C02041 V=800.0 PL=0
MOVL C02042 V=800.0 PL=0
MOVL C02043 V=800.0 PL=0
MOVL C02044 V=800.0 PL=0
MOVL C02045 V=800.0 PL=0
MOVL C02046 V=800.0 PL=0
MOVL C02047 V=800.0 PL=0
MOVL C02048 V=800.0 PL=0
MOVL C02049 V=800.0 PL=0
MOVL C02050 V=800.0 PL=0
MOVL C02051 V=800.0 PL=0
MOVL C02052 V=800.0 PL=0
MOVL C02053 V=800.0 PL=0
MOVL C02054 V=800.0 PL=0
MOVL C02055 V=800.0 PL=0
MOVL C02056 V=800.0 PL=0
MOVL C02057 V=800.0 PL=0
MOVL C02058 V=800.0 PL=0
MOVL C02059 V=800.0 PL=0
MOVL C02060 V=800.0 PL=0
MOVL C02061 V=800.0 PL=0
MOVL C02062 V=800.0 PL=0
MOVL C02063 V=800.0 PL=0
MOVL C02064 V=800.0 PL=0
MOVL C02065 V=800.0 PL=0
MOVL C02066 V=800.0 PL=0
MOVL C02067 V=800.0 PL=0
MOVL C02068 V=800.0 PL=0
MOVL C02069 V=800.0 PL=0
MOVL C02070 V=800.0 PL=0
MOVL C02071 V=800.0 PL=0
MOVL C02072 V=800.0 PL=0
MOVL C02073 V=800.0 PL=0
MOVL C02074 V=800.0 PL=0
MOVL C02075 V=800.0 PL=0
MOVL C02076 V=800.0 PL=0
MOVL C02077 V=800.0 PL=0
MOVL C02078 V=800.0 PL=0
MOVL C02079 V=800.0 PL=0
MOVL C02080 V=800.0 PL=0
MOVL C02081 V=800.0 PL=0
MOVL C02082 V=800.0 PL=0
MOVL C02083 V=800.0 PL=0
MOVL C02084 V=800.0 PL=0
MOVL C02085 V=800.0 PL=0
MOVL C02086 V=800.0 PL=0
MOVL C02087 V=800.0 PL=0
MOVL C02088 V=800.0 PL=0
MOVL C02089 V=800.0 PL=0
MOVL C02090 V=800.0 PL=0
MOVL C02091 V=800.0 PL=0
MOVL C02092 V=800.0 PL=0
MOVL C02093 V=800.0 PL=0
MOVL C02094 V=800.0 PL=0
MOVL C02095 V=800.0 PL=0
MOVL C02096 V=800.0 PL=0
MOVL C02097 V=800.0 PL=0
MOVL C02098 V=800.0 PL=0
MOVL C02099 V=800.0 PL=0
MOVL C02100 V=800.0 PL=0
MOVL C02101 V=800.0 PL=0
MOVL C02102 V=800.0 PL=0
MOVL C02103 V=800.0 PL=0
MOVL C02104 V=800.0 PL=0
MOVL C02105 V=800.0 PL=0
MOVL C02106 V=800.0 PL=0
MOVL C02107 V=800.0 PL=0
MOVL C02108 V=800.0 PL=0
MOVL C02109 V=800.0 PL=0
MOVL C02110 V=800.0 PL=0
MOVL C02111 V=800.0 PL=0
MOVL C02112 V=800.0 PL=0
MOVL C02113 V=800.0 PL=0
MOVL C02114 V=800.0 PL=0
MOVL C02115 V=800.0 PL=0
MOVL C02116 V=800.0 PL=0
MOVL C02117 V=800.0 PL=0
MOVL C02118 V=800.0 PL=0
MOVL C02119 V=800.0 PL=0
MOVL C02120 V=800.0 PL=0
